_fbFileClose(
	sNetId:= , 
	hFile:=_fbFileOpen.hFile , 
	bExecute:= , 
	tTimeout:= , 
	bBusy=> , 
	bError=> , 
	nErrId=> );
	
A_Run();
A_Status();

ACTION A_Run:
{attribute'hide'}

IF NOT Execute THEN
	_iRun:=0;
END_IF

CASE _iRun OF
	0:
		Done:=FALSE;
		_fbFileOpen.bExecute:=FALSE;
		_fbFileClose.bExecute:=FALSE;
		_fbFileWrite.bExecute:=FALSE;
		IF Execute THEN
			_iRun:=100;
		END_IF
	100:
		_fbFileOpen.bExecute:=TRUE;
		IF _fbFileOpen.bBusy THEN
			_iRun:=200;
		END_IF
	200:
		IF NOT _fbFileOpen.bBusy  THEN
			_fbFileOpen.bExecute:=FALSE;
			_iRun:=300;
		END_IF

	300:
		_fbFileWrite.bExecute:=TRUE;
		IF _fbFileWrite.bBusy  THEN
			_iRun:=400;
		END_IF
	400:
		IF NOT _fbFileWrite.bBusy THEN
			_fbFileWrite.bExecute:=FALSE;
			_iRun:=500;
		END_IF
	500:
		_fbFileClose.bExecute:=TRUE;
		IF _fbFileClose.bBusy  THEN
			_iRun:=600;
		END_IF
	600:
		IF NOT _fbFileClose.bBusy THEN
			_fbFileClose.bExecute:=FALSE;
			_iRun:=700;
		END_IF
	700:
		Done:=TRUE;
		IF NOT Execute  THEN
			_iRun:=0;
		END_IF
END_CASE
END_ACTION

ACTION A_Status:
{attribute'hide'}

Busy:= _fbFileOpen.bBusy  OR _fbFileWrite.bBusy OR _fbFileClose.bBusy;

Error:=_fbFileOpen.bError OR _fbFileWrite.bError OR _fbFileClose.bError;
END_ACTION

END_FUNCTION_BLOCK

// File/POUs/FB_LogHelper_B
FUNCTION_BLOCK FB_LogHelper_B // 带缓存功能的Log文件写入
VAR_INPUT
	System:						REFERENCE TO ST_System;
	FliePath:					STRING;// 文件夹路径					
	Message:					WSTRING(255);// 写入信息
END_VAR
VAR_OUTPUT
END_VAR
VAR
	_fbFileLog:					FB_LogHelper;
	_fbFifo:					FB_MemRingBuffer;
	_sFifoWrite:				WSTRING(255);
	_sFifoRead:					WSTRING(255);
	_arrFifoBuffer:				ARRAY[0..1000] OF WSTRING(255);
	_iFifoCount:				UDINT;
	_tonWrite:					TON;
	_fbDirectoryHelper:			FB_DirectoryHelper1;
END_VAR

IF _fbFifo.nCount>0 AND NOT _fbFileLog.Execute  AND NOT _fbFileLog.Done  AND NOT _tonWrite.Q THEN
	_sFifoRead:="";
	_iFifoCount:=_fbFifo.nCount;
	_fbFifo.A_RemoveHead();
	_fbFileLog.Message:=_sFifoRead;
	_fbFileLog.Execute:=TRUE;
END_IF
IF  _fbFileLog.Done OR _fbFileLog.Error THEN
	_fbFileLog.Execute:=FALSE;
END_IF


_fbDirectoryHelper(
	Execute:=TRUE , 
	Command:=E_Directory.Create , 
	FolderPath:=FliePath , 
	Busy=> , 
	Error=> , 
	Done=> );

_fbFileLog(
	Execute:= , 
	FilePath:=CONCAT(CONCAT(CONCAT(FliePath,'\'),System.stSystemDate.sDateDay),'.txt') , 
	Message:= , 
	Done=> , 
	Busy=> , 
	Error=> , 
	ErrId=> );
	
_fbFifo(
	pWrite:=ADR(_sFifoWrite) , 
	cbWrite:=SIZEOF(_sFifoWrite) , 
	pRead:=ADR(_sFifoRead) , 
	cbRead:=SIZEOF(_sFifoRead) , 
	pBuffer:=ADR(_arrFifoBuffer) , 
	cbBuffer:=SIZEOF(_arrFifoBuffer) , 
	bOk=> , 
	nCount=> , 
	cbSize=> , 
	cbReturn=> );
	
_tonWrite(IN:=_fbFifo.nCount=_iFifoCount AND NOT _fbFifo.nCount<>0  , PT:=T#2S , Q=> , ET=> );

ACTION A_AddTail:
_sFifoWrite:=Message;
_fbFifo.A_AddTail();
END_ACTION

END_FUNCTION_BLOCK

// File/POUs/FB_LogHelper_E
FUNCTION_BLOCK FB_LogHelper_E// 英文Log文件写入
VAR_INPUT
	Execute:				BOOL;
	FilePath:				STRING;
	Message:				STRING(1000);
END_VAR
VAR_OUTPUT
	Done:					BOOL;
	Busy:					BOOL;
	Error:					BOOL;
	ErrId:					INT;// 暂未使用
END_VAR
VAR
	_iRun:					INT;
	_fbFileOpen:			FB_FileOpen;
	_fbFileWrite:			FB_FileWrite;
	_fbFileClose:			FB_FileClose;
	_sTempString:			STRING(1000);
	_arrTemp:				ARRAY[0..1] OF STRING(1000);
	_sSeparator:			STRING;
END_VAR

_fbFileOpen(
	sNetId:= , 
	sPathName:=FilePath , 
	nMode:=FOPEN_MODEAPPEND , 
	ePath:= , 
	bExecute:= , 
	tTimeout:= , 
	bBusy=> , 
	bError=> , 
	nErrId=> , 
	hFile=> );

_arrTemp[0]:=Message;
_arrTemp[1]:='$N';
_sTempString:=F_Join_L(ADR(_arrTemp),SIZEOF(_arrTemp[0]),1,ADR(_sSeparator),SIZEOF(_sSeparator));

_fbFileWrite(
	sNetId:= , 
	hFile:=_fbFileOpen.hFile , 
	pWriteBuff:=ADR(_sTempString) , 
	cbWriteLen:=F_LEN(ADR(_sTempString)), 
	bExecute:= , 
	tTimeout:= , 
	bBusy=> , 
	bError=> , 
	nErrId=> , 
	cbWrite=> );

_fbFileClose(
	sNetId:= , 
	hFile:=_fbFileOpen.hFile , 
	bExecute:= , 
	tTimeout:= , 
	bBusy=> , 
	bError=> , 
	nErrId=> );
	
A_Run();
A_Status();

ACTION A_Run:
{attribute'hide'}

IF NOT Execute THEN
	_iRun:=0;
END_IF

CASE _iRun OF
	0:
		Done:=FALSE;
		_fbFileOpen.bExecute:=FALSE;
		_fbFileClose.bExecute:=FALSE;
		_fbFileWrite.bExecute:=FALSE;
		IF Execute THEN
			_iRun:=100;
		END_IF
	100:
		_fbFileOpen.bExecute:=TRUE;
		IF _fbFileOpen.bBusy THEN
			_iRun:=200;
		END_IF
	200:
		IF NOT _fbFileOpen.bBusy  THEN
			_fbFileOpen.bExecute:=FALSE;
			_iRun:=300;
		END_IF

	300:
		_fbFileWrite.bExecute:=TRUE;
		IF _fbFileWrite.bBusy  THEN
			_iRun:=400;
		END_IF
	400:
		IF NOT _fbFileWrite.bBusy THEN
			_fbFileWrite.bExecute:=FALSE;
			_iRun:=500;
		END_IF
	500:
		_fbFileClose.bExecute:=TRUE;
		IF _fbFileClose.bBusy  THEN
			_iRun:=600;
		END_IF
	600:
		IF NOT _fbFileClose.bBusy THEN
			_fbFileClose.bExecute:=FALSE;
			_iRun:=700;
		END_IF
	700:
		Done:=TRUE;
		IF NOT Execute  THEN
			_iRun:=0;
		END_IF
END_CASE
END_ACTION

ACTION A_Status:
{attribute'hide'}

Busy:= _fbFileOpen.bBusy  OR _fbFileWrite.bBusy OR _fbFileClose.bBusy;

Error:=_fbFileOpen.bError OR _fbFileWrite.bError OR _fbFileClose.bError;
END_ACTION

END_FUNCTION_BLOCK

// Regex/F_Join_L
FUNCTION F_Join_L:STRING(2000)
VAR_INPUT
	In:						POINTER TO BYTE;// 拼接字符串数组
	OneLength:				UDINT;//Sizeof(In[0])
	Count:					INT;// 数组长度
	Separator:				POINTER TO BYTE;// 分隔符
	SeparatorLength:		UDINT;//Sizeof(SeparatorLength)
END_VAR
VAR
	_i:						LINT;// 输入字符串数组循环
	_t:						LINT;// 单个输入字符串循环
	_f:						LINT;// 输出元素索引
	_a:						LINT;// 
	_pTemp:					POINTER TO BYTE;
	_iTemplen:				UINT;
END_VAR

_pTemp:=ADR(F_Join_L);
_iTemplen:=SIZEOF(F_Join_L);

FOR _i:=0 TO Count BY 1 DO
	FOR _t:=(_i*OneLength) TO (OneLength-1)+(OneLength*_i) BY 1 DO
		IF _f>=_iTemplen-1 THEN RETURN; END_IF;
		IF In[_t]=0 THEN EXIT; END_IF;
		_pTemp[_f]:=In[_t];
		_f:=_f+1;
	END_FOR
	IF _i=Count THEN
		EXIT;
	END_IF
	FOR _a:=0 TO SeparatorLength-1 BY 1 DO
		IF _f>=_iTemplen-1 THEN RETURN; END_IF;
		IF Separator[_a]=0 THEN EXIT; END_IF;
		_pTemp[_f]:=Separator[_a];
		_f:=_f+1;
	END_FOR
END_FOR
_pTemp[_f]:=0;

END_FUNCTION

// File/POUs/FB_LogHelper_E_B
FUNCTION_BLOCK FB_LogHelper_E_B// 英文带缓存的Log文件写入
VAR_INPUT
	System:						REFERENCE TO ST_System;
	DocumentPath:				STRING;// 文件夹路径					
	Message:					STRING(1000);// 写入信息
	FilePath:					STRING(1000);// 文件路径(当文件路径为空时 则按文件夹路路径自动生成文件)
END_VAR
VAR_OUTPUT
END_VAR
VAR
	_fbFileLog:					FB_LogHelper_E;
	_fbFifo:					FB_MemRingBuffer;
	_sFifoWrite:				STRING(1000);
	_sFifoRead:					STRING(1000);
	_arrFifoBuffer:				ARRAY[0..1000] OF STRING(1000);
	_iFifoCount:				UDINT;
	_tonWrite:					TON;
	_fbDirectoryHelper:			FB_DirectoryHelper;
END_VAR

IF _fbFifo.nCount>0 AND NOT _fbFileLog.Execute  AND NOT _fbFileLog.Done  AND NOT _tonWrite.Q THEN
	_sFifoRead:='';
	_iFifoCount:=_fbFifo.nCount;
	_fbFifo.A_RemoveHead();
	_fbFileLog.Message:=_sFifoRead;
	_fbFileLog.Execute:=TRUE;
END_IF
IF  _fbFileLog.Done OR _fbFileLog.Error THEN
	_fbFileLog.Execute:=FALSE;
END_IF

_fbDirectoryHelper(
	Execute:=TRUE , 
	Command:=E_Directory.Create , 
	DirectoryPath:=FilePath , 
	Busy=> , 
	Error=> , 
	Done=> );

_fbFileLog(
	Execute:= , 
	FilePath:=SEL(FilePath='',FilePath,CONCAT(CONCAT(CONCAT(DocumentPath,'\'),System.stSystemDate.sDateDay),'.txt')), 
	Message:= , 
	Done=> , 
	Busy=> , 
	Error=> , 
	ErrId=> );
	
_fbFifo(
	pWrite:=ADR(_sFifoWrite) , 
	cbWrite:=SIZEOF(_sFifoWrite) , 
	pRead:=ADR(_sFifoRead) , 
	cbRead:=SIZEOF(_sFifoRead) , 
	pBuffer:=ADR(_arrFifoBuffer) , 
	cbBuffer:=SIZEOF(_arrFifoBuffer) , 
	bOk=> , 
	nCount=> , 
	cbSize=> , 
	cbReturn=> );
	
_tonWrite(IN:=_fbFifo.nCount=_iFifoCount AND NOT _fbFifo.nCount<>0  , PT:=T#2S , Q=> , ET=> );

ACTION A_AddTail:
_sFifoWrite:=Message;
_fbFifo.A_AddTail();
END_ACTION

END_FUNCTION_BLOCK

// File/POUs/FB_LogHelper1
FUNCTION_BLOCK FB_LogHelper1
VAR_INPUT
	FilePath:				STRING;// 文件路径
	pBuffer:				PVOID;// 缓存数据区
	cbBuffer:				UDINT;// sizfof(cbBuffer)
	Message:				PVOID;// 写入信息
END_VAR
VAR_OUTPUT
END_VAR
VAR
	_sFifoRead:				STRING(1000);
	_iFifoCount:			UDINT;
	_fbFileHelper:			FB_FileHelper;
	_fbFifo:				FB_MemRingBuffer;
END_VAR

_fbFifo(
	pWrite:= , 
	cbWrite:= , 
	pRead:=ADR(_sFifoRead) , 
	cbRead:=SIZEOF(_sFifoRead) , 
	pBuffer:=pBuffer , 
	cbBuffer:=cbBuffer , 
	bOk=> , 
	nCount=> , 
	cbSize=> , 
	cbReturn=> );
_fbFileHelper(
	Read:= , 
	WriteAllText:= , 
	AppendAllText:= , 
	FilePath:=FilePath , 
	Buffer:=ADR(_sFifoRead) , 
	BufferLen:=F_LEN(ADR(_sFifoRead)) , 
	TimeOut:= , 
	Busy=> , 
	Error=> , 
	Done=> );
	
	
IF _fbFifo.nCount>0 AND NOT _fbFileHelper.AppendAllText THEN
	_sFifoRead:='';
	_fbFifo.A_RemoveHead();
	_fbFileHelper.AppendAllText:=TRUE;
END_IF
IF  _fbFileHelper.Done THEN
	_fbFileHelper.AppendAllText:=FALSE;
END_IF

METHOD M_AddTail : BOOL
VAR_INPUT
END_VAR
_fbFifo.pWrite:=Message;
_fbFifo.cbWrite:=F_LEN(Message);
_fbFifo.A_AddTail();
M_AddTail:=TRUE;
END_METHOD

END_FUNCTION_BLOCK

// Hive/POUs/FB_Hive
FUNCTION_BLOCK FB_Hive
VAR_INPUT
	System:				 	 REFERENCE TO ST_System;
	Error:				  	 REFERENCE TO ST_Error;
	Hive:					 REFERENCE TO ST_Hive;
	Data:					 REFERENCE TO ST_HiveData;
END_VAR
VAR_OUTPUT
END_VAR
VAR
	_arrFbHttpClient:		ARRAY[0..3] OF FB_HttpClient;
	_arrHttpClient:			ARRAY[0..3] OF ST_HttpClient;
	_arrHttpClientData:		ARRAY[0..3] OF ST_HttpClientData;
	_i:						INT;
	_eHiveState:			E_HiveState:=E_HiveState.None;
	_iStateRun:				INT;
	_iDataRun:				INT;
	_sDataTime:				STRING;
	
	_arrErrorTemp:			ARRAY[0..100] OF STRING;
	_arrErrorCode:			ARRAY[0..100] OF STRING;
	_arrErrorMessage:		ARRAY[0..100] OF STRING;
	_iErrorCount:			INT:=0;
	_sErrorMessageTemp:		STRING(1000);
	
	_arrTon:				ARRAY[0..10] OF TON;
	
	_iRunCount:				INT:=0;
	
	_iModeRun:				INT;
	_bFirstRun:				BOOL:=TRUE;
END_VAR

IF _iRunCount<3 THEN
	_iRunCount:=_iRunCount+1;
	RETURN;
END_IF
IF  _bFirstRun THEN
	A_Init();
END_IF



IF Hive.stControl.bDataEnable THEN
	_arrFbHttpClient[0](System:=System , Error:=Error , HttpClient:=_arrHttpClient[0] , Data:=_arrHttpClientData[0] );
END_IF

IF Hive.stControl.bDataEnable THEN
	_arrFbHttpClient[1](System:=System , Error:=Error , HttpClient:=_arrHttpClient[1] , Data:=_arrHttpClientData[1] );
END_IF

IF Hive.stControl.bStateEnable THEN
	_arrFbHttpClient[2](System:=System , Error:=Error , HttpClient:=_arrHttpClient[2] , Data:=_arrHttpClientData[2] );
END_IF

IF Hive.stControl.bDataEnable THEN
	_arrFbHttpClient[3](System:=System , Error:=Error , HttpClient:=_arrHttpClient[3] , Data:=_arrHttpClientData[3] );
END_IF



//2020-08-27T00:01:29.51+0800
_sDataTime:=M_DateTime();
A_Data();
A_Mode();
A_State();
A_Ton();

_bFirstRun:=FALSE;

ACTION A_Data:
{attribute'hide'}

IF System.stInput.bReset OR NOT  Hive.stControl.bDataEnable THEN
	_iDataRun:=0;
END_IF

CASE _iDataRun OF
	0:
		Hive.stSendDataState.bDone:=FALSE;
		Hive.stSendDataState.bBusy:=FALSE;
		Hive.stSendDataState.bError:=FALSE;
		_arrHttpClient[0].stControl.eRequest:=E_HttpRequestOrder.None;
		IF Hive.stControl.bSendData AND Hive.stControl.bDataEnable THEN
			_iDataRun:=100;
		END_IF;
	100:
		Hive.stSendDataState.bBusy:=TRUE;
		_arrHttpClient[0].stControl.sRequestData:=M_Data();
		_iDataRun:=200;
	200:
		_arrHttpClient[0].stControl.eRequest:=E_HttpRequestOrder.POST;
		IF _arrHttpClient[0].stStatus.bDone OR _arrTon[2].Q  THEN
			_arrHttpClient[0].stControl.eRequest:=E_HttpRequestOrder.None;
			_iDataRun:=300;
		END_IF
	300:
		IF  _arrTon[2].Q THEN
			Hive.stSendDataState.bError:=TRUE;
		END_IF;
		_iDataRun:=400;
	400:
		Hive.stSendDataState.bBusy:=FALSE;
		Hive.stSendDataState.bDone:=TRUE;
		IF NOT  Hive.stControl.bSendData AND NOT System.stMode.bStop THEN
			Hive.stSendDataState.bDone:=FALSE;
			_iDataRun:=0;
		END_IF
END_CASE
END_ACTION

ACTION A_Init:
{attribute'hide'}

_arrHttpClient[0].arrInfo[E_Language.Chinese].sName:="Hive_Data";
_arrHttpClient[0].arrInfo[E_Language.English].sName:="Hive_Data";
_arrHttpClient[0].arrInfo[E_Language.Hindi].sName:="Hive_Data";
_arrHttpClient[0].arrInfo[E_Language.Vietnamese].sName:="Hive_Data";
_arrHttpClientData[0].iPort:=Data.stDataAddress.iPort;
_arrHttpClientData[0].iTimeOut:=Data.iTimeOut;
_arrHttpClientData[0].sIP:=Data.stDataAddress.sIP;
_arrHttpClientData[0].sUri:=Data.stDataAddress.sUri;

_arrHttpClient[1].arrInfo[E_Language.Chinese].sName:="Hive_Mode";
_arrHttpClient[1].arrInfo[E_Language.English].sName:="Hive_Mode";
_arrHttpClient[1].arrInfo[E_Language.Hindi].sName:="Hive_Mode";
_arrHttpClient[1].arrInfo[E_Language.Vietnamese].sName:="Hive_Mode";
_arrHttpClientData[1].iPort:=Data.stModeAddressOn.iPort;
_arrHttpClientData[1].iTimeOut:=Data.iTimeOut;
_arrHttpClientData[1].sIP:=Data.stModeAddressOn.sIP;
_arrHttpClientData[1].sUri:=Data.stModeAddressOn.sUri;

_arrHttpClient[2].arrInfo[E_Language.Chinese].sName:="Hive_State";
_arrHttpClient[2].arrInfo[E_Language.English].sName:="Hive_State";
_arrHttpClient[2].arrInfo[E_Language.Hindi].sName:="Hive_State";
_arrHttpClient[2].arrInfo[E_Language.Vietnamese].sName:="Hive_State";
_arrHttpClientData[2].iPort:=Data.stStateAddress.iPort;
_arrHttpClientData[2].iTimeOut:=Data.iTimeOut;
_arrHttpClientData[2].sIP:=Data.stStateAddress.sIP;
_arrHttpClientData[2].sUri:=Data.stStateAddress.sUri;

_arrHttpClient[3].arrInfo[E_Language.Chinese].sName:="Hive_Mode";
_arrHttpClient[3].arrInfo[E_Language.English].sName:="Hive_Mode";
_arrHttpClient[3].arrInfo[E_Language.Hindi].sName:="Hive_Mode";
_arrHttpClient[3].arrInfo[E_Language.Vietnamese].sName:="Hive_Mode";
_arrHttpClientData[3].iPort:=Data.stModeAddressOff.iPort;
_arrHttpClientData[3].iTimeOut:=Data.iTimeOut;
_arrHttpClientData[3].sIP:=Data.stModeAddressOff.sIP;
_arrHttpClientData[3].sUri:=Data.stModeAddressOff.sUri;
END_ACTION

ACTION A_Mode:
{attribute'hide'}

IF  _arrTon[3].Q OR _arrTon[4].Q THEN
	_iModeRun:=0;
END_IF

CASE _iModeRun OF
	0:
		_arrTon[3].IN:=_arrTon[4].IN:=FALSE;
		_arrHttpClient[1].stControl.eRequest:=E_HttpRequestOrder.None;
		_arrHttpClient[3].stControl.eRequest:=E_HttpRequestOrder.None;
		IF Hive.stControl.bModeLogin AND Hive.stControl.bModeEnable THEN
			_iModeRun:=100;
		END_IF
	100:
		_arrHttpClient[1].stControl.sRequestData:=M_ModeOn();
		_iModeRun:=200;
	200:
		_arrTon[3].IN:=TRUE;
		_arrHttpClient[1].stControl.eRequest:=E_HttpRequestOrder.POST;
		IF _arrHttpClient[1].stStatus.bDone THEN
			_arrHttpClient[1].stControl.eRequest:=E_HttpRequestOrder.None;
			_iModeRun:=300;
		END_IF
	300:
		IF NOT Hive.stControl.bModeLogin THEN
			_iModeRun:=400;
		END_IF
	400:
		_arrHttpClient[3].stControl.sRequestData:=M_ModeOff();
		_iModeRun:=500;
	500:
		_arrTon[4].IN:=TRUE;
		_arrHttpClient[3].stControl.eRequest:=E_HttpRequestOrder.POST;
		IF _arrHttpClient[3].stStatus.bDone THEN
			_arrHttpClient[3].stControl.eRequest:=E_HttpRequestOrder.None;
			_iModeRun:=0;
		END_IF
END_CASE
END_ACTION

ACTION A_State:
{attribute'hide'}

IF System.stMode.bAutoRunning OR System.stMode.bHoming THEN
	_eHiveState:=E_HiveState.Running;
END_IF;

IF System.stMode.bIdle OR System.stMode.bNone THEN
	_eHiveState:=E_HiveState.Idle;
END_IF;

IF System.stMode.arrAlarm[1] OR  System.stMode.arrAlarm[2] OR System.stMode.arrAlarm[3] THEN
	_eHiveState:=E_HiveState.UnplannedDown;
END_IF;

IF System.stMode.bManual THEN
	_eHiveState:=E_HiveState.Engineering;
END_IF;

IF Hive.stControl.bPlannedDown THEN
	_eHiveState:=E_HiveState.PlannedDown;
END_IF;


IF _arrTon[1].Q OR NOT Hive.stControl.bStateEnable THEN
	_iStateRun:=0;
END_IF; 

CASE _iStateRun OF
	0:
		_arrTon[0].IN:=FALSE;
		_arrHttpClient[2].stControl.eRequest:=E_HttpRequestOrder.None;
		IF _eHiveState <> Hive.eState AND Hive.stControl.bStateEnable AND NOT _arrTon[1].Q THEN
			_iStateRun:=100;
		END_IF;
	100:
		CASE _eHiveState OF
			0:
				_iStateRun:=0;
			1,2,3,4:
				_iStateRun:=200;
			5:
				_iStateRun:=500;
		END_CASE
	200:
		_arrHttpClient[2].stControl.sRequestData:=M_State(_eHiveState,'');
		_iStateRun:=1000;
	500:
		FOR _i:=0 TO 100 BY 1 DO
			_arrErrorTemp[_i]:='';
			_arrErrorCode[_i]:='';
			_arrErrorMessage[_i]:='';
			_iErrorCount:=0;
		END_FOR
		_iStateRun:=510;
	510:// 报警信息为: 报警文本;报警代码
		FOR _i:=0 TO Error.stNow.iCount BY 1 DO
			IF STRING_TO_INT(Error.stNow.arrInfo[_i].sLevel)<=3 AND Error.stNow.arrInfo[_i].sLevel<>'' THEN
				_sErrorMessageTemp:=WSTRING_TO_STRING(Error.stNow.arrInfo[_i].arrMessage[Data.eLanguage]);
				F_Split(ADR(_sErrorMessageTemp),ADR(';'),ADR(_arrErrorTemp),SIZEOF(_arrErrorTemp[0]),SIZEOF(_arrErrorTemp));
				EXIT;
			END_IF
		END_FOR
		_iStateRun:=515;
	515:
		_arrErrorMessage[_iErrorCount]:=_arrErrorTemp[0];
		_arrErrorCode[_iErrorCount]:=_arrErrorTemp[1];
		_iStateRun:=520;
	520:
		_arrErrorTemp[0]:=CONCAT(CONCAT(CONCAT(CONCAT(CONCAT('$R"code": "',_arrErrorCode[_iErrorCount]),'",'),'$R"error_message" : "'),_arrErrorMessage[_iErrorCount]),'",$R');
		_arrHttpClient[2].stControl.sRequestData:=M_State(_eHiveState,_arrErrorTemp[0]);
		_iErrorCount:=_iErrorCount+1;
		_iStateRun:=1000;
	1000:
		_arrTon[0].IN:=TRUE;
		_arrHttpClient[2].stControl.eRequest:=E_HttpRequestOrder.POST;
		IF _arrHttpClient[2].stStatus.bDone THEN
			_arrHttpClient[2].stControl.eRequest:=E_HttpRequestOrder.None;
			_iStateRun:=1100;
		END_IF
	1100:
		IF NOT _arrTon[0].Q THEN
			 Hive.eState:=_eHiveState;
		END_IF
		_iStateRun:=0;
END_CASE
END_ACTION

ACTION A_Ton:
{attribute'hide'}

_arrTon[0](IN:= , PT:=UINT_TO_TIME(Data.iTimeOut) , Q=> , ET=> );// State处理耗时
_arrTon[1](IN:= _iStateRun<>0, PT:=UINT_TO_TIME(Data.iTimeOut+1000), Q=> , ET=> );// State运行耗时

_arrTon[2](IN:=Hive.stSendDataState.bBusy , PT:=UINT_TO_TIME(Data.iTimeOut+500) , Q=> , ET=> );// Data处理耗时

_arrTon[3](IN:= , PT:=UINT_TO_TIME(Data.iTimeOut+500) , Q=> , ET=> );//ModeOn处理耗时
_arrTon[4](IN:= , PT:=UINT_TO_TIME(Data.iTimeOut+500) , Q=> , ET=> );//ModeOff处理耗时
END_ACTION

{attribute'hide'}
METHOD M_Data : STRING(2000)
VAR_INPUT
END_VAR
VAR
	_t:						INT;
	_arrTemp:				ARRAY[0..400] OF STRING;
	_iCount:				INT;
	_temp:					POINTER TO BYTE;
END_VAR


_arrTemp[0]:='{';
_arrTemp[1]:=CONCAT(CONCAT('"unit_sn": "',Hive.stControl.stMachineData.sUnit_sn),'",');
_arrTemp[2]:='"serials": {';
_arrTemp[3]:=CONCAT(CONCAT('"carrier_sn": "',Hive.stControl.stMachineData.sCarrier_sn),'",');
_arrTemp[4]:=CONCAT(CONCAT('"wip_serials" : ["',Hive.stControl.stMachineData.sWip_serials),'"]},');
_arrTemp[5]:=CONCAT(CONCAT('"pass": "',BOOL_TO_STRING( Hive.stControl.stMachineData.bPass)),'",');
_arrTemp[6]:=CONCAT(CONCAT('"input_time": "',Hive.stControl.stMachineData.sInput_time),'",');
_arrTemp[7]:=CONCAT(CONCAT('"output_time": "',Hive.stControl.stMachineData.sOutput_time),'",');
_arrTemp[8]:='"data": {';
_iCount:=8;
FOR _t:=0 TO Hive.stControl.stMachineData.iDataCount-1 BY 1 DO
	IF Hive.stControl.stMachineData.arrDataName[_t]<>'' THEN
		_arrTemp[9+_t]:=CONCAT(CONCAT(CONCAT(CONCAT('"',Hive.stControl.stMachineData.arrDataName[_t]),'":"'),Hive.stControl.stMachineData.arrDataValue[_t]),'",');
		_iCount:=_iCount+1;
	END_IF;
END_FOR
IF _iCount>8 THEN
	_temp:=ADR(_arrTemp[_iCount]);
	_temp[F_LEN(ADR(_arrTemp[_iCount]))-1]:=0;
END_IF
_arrTemp[_iCount+1]:='}$R}';

M_Data:=F_Join_L(ADR(_arrTemp),SIZEOF(_arrTemp[0]),_iCount+1,ADR('$R'),SIZEOF('$R'));
END_METHOD

{attribute'hide'}
METHOD M_DateTime : string
VAR_INPUT
END_VAR


M_DateTime:=CONCAT(CONCAT(CONCAT(CONCAT(CONCAT(CONCAT(CONCAT(CONCAT(CONCAT(CONCAT(CONCAT(CONCAT(CONCAT(CONCAT(INT_TO_STRING(System.stSystemDate.iYear),'-'),M_Join0(system.stSystemDate.iMonth)),'-'),M_Join0(system.stSystemDate.iDay)),'T'),M_Join0(system.stSystemDate.iHour)),':'),M_Join0(system.stSystemDate.iMinute)),':'),M_Join0(system.stSystemDate.iSecond)),'.'),INT_TO_STRING(System.stSystemDate.iMilliseconds)),'+'),'0800');
END_METHOD

{attribute'hide'}
METHOD M_Join0 : STRING
VAR_INPUT
	In:					INT;
END_VAR


M_Join0:=SEL(In<10,INT_TO_STRING(In),CONCAT('0',INT_TO_STRING(In)));
END_METHOD

{attribute'hide'}
METHOD M_ModeOff : STRING(2000)
VAR_INPUT
END_VAR
VAR
	_arrTemp:				ARRAY[0..2] OF STRING(1000);
	_arrTemp1:				ARRAY[0..100] OF STRING;
	_iCount:				INT:=0;
	_t:						INT;
END_VAR


FOR _t:=0 TO Hive.stControl.iActivityCount-1 BY 1 DO
	IF Hive.stControl.arrActivity[_t]<>'' THEN
		_arrTemp1[_t]:=CONCAT(CONCAT('"', Hive.stControl.arrActivity[_t]),'"');
		_iCount:=_iCount+1;
	END_IF
END_FOR

_arrTemp[0]:=CONCAT(CONCAT('{$R"state_time": "',_sDataTime),'",$R"data": {$R"activity" : [');
_arrTemp[1]:=F_Join_L(ADR(_arrTemp1),SIZEOF(_arrTemp1[0]),_iCount-1,ADR(','),SIZEOF(','));;
_arrTemp[2]:= CONCAT(CONCAT('],$R"session_token": "',Hive.stControl.sSession_token),'"$R}$R}');


M_ModeOff:=F_Join_L(ADR(_arrTemp),SIZEOF(_arrTemp[0]),2,ADR('$R'),SIZEOF('$R'));
END_METHOD

{attribute'hide'}
METHOD M_ModeOn : STRING(2000)
VAR_INPUT
END_VAR
VAR
	_arrTemp:				ARRAY[0..10] OF STRING(100);
END_VAR


_arrTemp[0]:='{';
_arrTemp[1]:=CONCAT(CONCAT('"state_time": "',_sDataTime),'",');
_arrTemp[2]:='"data": {';
_arrTemp[3]:= CONCAT(CONCAT('"session_token": "',Hive.stControl.sSession_token),'"');
_arrTemp[4]:='}';
_arrTemp[5]:='}';

M_ModeOn:=F_Join_L(ADR(_arrTemp),SIZEOF(_arrTemp[0]),5,ADR('$R'),SIZEOF('$R'));
END_METHOD

{attribute'hide'}
METHOD M_State : STRING(2000)
VAR_INPUT
	State:					INT;
	Data:					STRING(1000);
END_VAR
VAR
	_arrTemp:				ARRAY[0..100] OF STRING(255);
END_VAR


_arrTemp[0]:='{';
_arrTemp[1]:=CONCAT(CONCAT('"machine_state":',INT_TO_STRING(State)),',');
_arrTemp[2]:=CONCAT(CONCAT('"state_change_time": "',_sDataTime),'",');
_arrTemp[3]:=CONCAT(CONCAT('"data": {',Data),'}');
_arrTemp[4]:='}';
M_State:=F_Join_L(ADR(_arrTemp),SIZEOF(_arrTemp[0]),4,ADR('$R'),SIZEOF('$R'));
END_METHOD

END_FUNCTION_BLOCK

// Http/POUs/FB_HttpClient
FUNCTION_BLOCK FB_HttpClient
VAR_INPUT
	System:						REFERENCE TO ST_System;
	Error:						REFERENCE TO ST_Error;
	HttpClient:					REFERENCE TO ST_HttpClient;
	Data:						REFERENCE TO ST_HttpClientData;
END_VAR
VAR_OUTPUT
END_VAR
VAR
	_fbIotHttpClient:					FB_IotHttpClient();
	_fbIotHttpRequest:					FB_IotHttpRequest();
	_fbIotHttpHeaderFieldMap:			FB_IotHttpHeaderFieldMap();
	_run:								INT;
	_arrFbErrorTag:						ARRAY[0..2] OF FB_ErrorTag;
	_i:									INT;
	_bFistRun:							BOOL:=TRUE;
END_VAR

HttpClient.sName:=HttpClient.arrInfo[System.stMode.eLanguage].sName;

_fbIotHttpClient.sHostName:=Data.sIP;
_fbIotHttpClient.nHostPort:=Data.iPort;
_fbIotHttpClient.Execute();

IF System.stInput.bReset THEN
	HttpClient.stControl.eRequest:=E_HttpRequestOrder.None;
	_run:=0;
END_IF;

IF _bFistRun THEN
	A_Init();
END_IF

A_Run();

A_Error();

_bFistRun:=FALSE;

ACTION A_Error:
{attribute'hide'}

_arrFbErrorTag[0](
	System:=System , 
	Error:=Error , 
	Enable:=_fbIotHttpClient.bError OR _fbIotHttpRequest.bError OR _fbIotHttpHeaderFieldMap.bError , 
	Message:=, 
	Level:=5 , 
	Position:=WCONCAT("FB_HttpClient:",HttpClient.arrInfo[E_Language.Chinese].sName) , 
	ErrorTime:= , 
	Language:= , 
	Erroring=>HttpClient.stStatus.bError,
	ID:=HttpClient.ID,
	Category:=E_ErrorCategory.Http,
	InfoIndex:=0);

	
_arrFbErrorTag[1](
	System:=System , 
	Error:=Error , 
	Enable:=HttpClient.stStatus.bBusy, 
	Message:="Http通信超时" , 
	Level:=5 , 
	Position:=WCONCAT("FB_HttpClient:",HttpClient.arrInfo[E_Language.Chinese].sName) , 
	ErrorTime:=UINT_TO_TIME(Data.iTimeOut), 
	Language:= , 
	Erroring=> HttpClient.stStatus.bErrorTimeOut,
	ID:=HttpClient.ID,
	Category:=E_ErrorCategory.Http,
	InfoIndex:=1);
END_ACTION

ACTION A_Init:
{attribute'hide'}
	HttpClient.arrInfo[E_Language.Chinese].sError:="状态错误";
	HttpClient.arrInfo[E_Language.Chinese].sErrorTimeOut:="请求超时";
	
	HttpClient.arrInfo[E_Language.English].sError:="Status error";
	HttpClient.arrInfo[E_Language.English].sErrorTimeOut:="Request timeout";
	
	HttpClient.arrInfo[E_Language.Hindi].sError:="स्थिति गलत है";
	HttpClient.arrInfo[E_Language.Hindi].sErrorTimeOut:="अनुरोध समय पर बाहर";
	
	HttpClient.arrInfo[E_Language.Vietnamese].sError:="Lỗi trạng thái";
	HttpClient.arrInfo[E_Language.Vietnamese].sErrorTimeOut:="Yêu cầu thời gian chờ";

FOR _i:=0 TO E_Language.MaxCount BY 1 DO
	_arrFbErrorTag[0].Language[_i]:= WCONCAT(HttpClient.arrInfo[_i].sName,HttpClient.arrInfo[_i].sError);
	_arrFbErrorTag[1].Language[_i]:= WCONCAT(HttpClient.arrInfo[_i].sName,HttpClient.arrInfo[_i].sErrorTimeOut);
END_FOR;
END_ACTION

ACTION A_Run:
{attribute'hide'}

CASE _run OF
	0:
		HttpClient.stStatus.bBusy:=HttpClient.stStatus.bDone:=FALSE;
		IF HttpClient.stControl.eRequest<>E_HttpRequestOrder.None AND  NOT System.stMode.bStop THEN
			_run:=100;
		END_IF;
	100:
		HttpClient.stStatus.bBusy:=TRUE;
		CASE HttpClient.stControl.eRequest  OF
			E_HttpRequestOrder.GET:
				IF SendRequest(ETcIotHttpRequestType.HTTP_GET) THEN
					_run:=1000;
				END_IF
			E_HttpRequestOrder.POST:
				IF SendRequest(ETcIotHttpRequestType.HTTP_POST) THEN
					_run:=1000;
				END_IF
		END_CASE
	1000:
		IF NOT _fbIotHttpRequest.bBusy THEN
			HttpClient.stControl.sResponseData:='';
			_run:=1100;
		END_IF
	1100:
		IF _fbIotHttpRequest.nContentSize<>0 THEN
			_fbIotHttpRequest.GetContent(ADR(HttpClient.stControl.sResponseData),SIZEOF(HttpClient.stControl.sResponseData),TRUE);
		END_IF;
		_run:=1200;
	1200:
		HttpClient.stStatus.bBusy:=FALSE;
		HttpClient.stStatus.bDone:=TRUE;
		IF HttpClient.stControl.eRequest=E_HttpRequestOrder.None THEN
			HttpClient.stStatus.bDone:=FALSE;
			_run:=0;
		END_IF
END_CASE
END_ACTION

{attribute'hide'}
METHOD SendRequest : BOOL
VAR_INPUT
	 eRequestType : ETcIotHttpRequestType;
END_VAR
SendRequest:= _fbIotHttpRequest.SendRequest(sUri:=Data.sUri,fbClient:=_fbIotHttpClient,eRequestType:=eRequestType,pContent:=ADR(HttpClient.stControl.sRequestData),nContentSize:=F_LEN(ADR(HttpClient.stControl.sRequestData)),fbHeader:=_fbIotHttpHeaderFieldMap);
END_METHOD

END_FUNCTION_BLOCK

// Regex/F_Split
FUNCTION F_Split
VAR_INPUT
	In:							POINTER TO BYTE;// 要拆分的字符串
	Pattern:					POINTER TO BYTE;// 拆分规则
	Data:						POINTER TO BYTE;// 拆分分后 返回数组数据区
	OneLength:					UDINT;// Sizeof(Data[0])
	DataLength:					UDINT;// Sizeof(Data)
END_VAR
VAR
	_i:							LINT;// 拆分字符串 索引
	_t:							LINT;// 分隔符计数
	_tIdx:						LINT;// 分隔符位置 索引
	_f:							LINT;// 单个数据 索引
	_iLength:					LINT;// 分隔符与分割符 中间数据长度
	_tt:						LINT;// 分隔符计数
	_ttIdx:						LINT;// 分隔符位置 索引
	_iDataIdx:					LINT;// 数据数组 索引
	_x:							LINT;// 数据清空索引
	_y:							LINT;// 添加末尾数据索引
	_iPattern:					LINT;// 分隔符长度
	_idx:						LINT;// 末尾数据索引
	_bTemp:						BOOL;// 分隔符标志
END_VAR

FOR _x:=0 TO DataLength BY 1 DO
	Data[_x]:=0;
END_FOR
_iPattern:= F_LEN(Pattern);

WHILE In[_i]<> 0 DO
	WHILE _t<_iPattern AND In[_i]<> 0 DO
		_t:=SEL(In[_i]<>Pattern[_t],_t+1,0);
		_i:=_i+1;
	END_WHILE
	_bTemp:=_t>=_iPattern;
	_tIdx:=_i-1;
	FOR _f:=0 TO _iLength:=SEL(_ttIdx<>0,_tIdx-_ttIdx-1*_iPattern,_tIdx-_ttIdx-1*_iPattern-1) DO
		IF _iLength<0 OR _f>=OneLength OR NOT _bTemp THEN EXIT; END_IF;
		Data[_f+_iDataIdx*OneLength]:=In[SEL(_ttIdx<>0,_ttIdx+_f,_ttIdx+_f+1)];
	END_FOR
	IF In[_i]= 0 THEN EXIT; END_IF;
	_iDataIdx:=_iDataIdx+1;
	
	
	WHILE _tt<_iPattern AND In[_i]<> 0 DO
		_tt:=SEL(In[_i]<>Pattern[_tt],_tt+1,0);
		_i:=_i+1;
	END_WHILE
	_bTemp:=_tt>=_iPattern;
	_ttIdx:=_i-1;
	FOR _f:=0 TO _iLength:=_ttIdx-_tIdx-1*_iPattern-1 DO
		IF _iLength<0 OR _f>=OneLength OR NOT _bTemp THEN EXIT; END_IF;
		Data[_f+_iDataIdx*OneLength]:=In[_tIdx+_f+1];
	END_FOR
	IF In[_i]= 0 THEN EXIT; END_IF;
	_iDataIdx:=_iDataIdx+1;
	
	_t:=_tt:=0;
END_WHILE

IF _tIdx=0 AND _ttIdx=0 THEN
	FOR _y:=0 TO OneLength-1 BY 1 DO
		IF In[_y]=0 THEN EXIT; END_IF;
		Data[_y]:=In[_y];
	END_FOR
ELSIF NOT _bTemp THEN
	_idx:=SEL(_tIdx<_ttIdx,_ttIdx,_tIdx);
	FOR _y:=0 TO ABS(_tIdx-_ttIdx)-1 BY 1 DO
		Data[_y+_iDataIdx*OneLength]:=In[_idx+1+_y];
	END_FOR
END_IF

END_FUNCTION

// Regex/M_Join0
FUNCTION M_Join0 : String
VAR_INPUT
	In:				INT;
END_VAR
VAR
END_VAR

M_Join0:=SEL(In<10,INT_TO_STRING(In),CONCAT('0',INT_TO_STRING(In)));

END_FUNCTION

// Hive/POUs/P_Hive
PROGRAM P_Hive
VAR
END_VAR

METHOD M_Data : STRING(2000)
VAR_INPUT
	sUnit_sn:				STRING;
	sCarrier_sn:			STRING;
	sWip_serials:			STRING;
	sPass:					STRING;
	sInput_time:			STRING;
	sOutput_time:			STRING;
	arrDataName:			POINTER TO STRING;
	arrDataValue:			POINTER TO STRING;
	iDataCount:				UINT;
END_VAR
VAR
	_t:						UINT;
	_arrTemp:				ARRAY[0..10] OF STRING(255);
	_temp:					POINTER TO BYTE;
	_sData:					ARRAY[0..2] OF STRING(2000);
END_VAR
_arrTemp[0]:='{';
_arrTemp[1]:=CONCAT(CONCAT('"unit_sn": "',sUnit_sn),'",');
_arrTemp[2]:='"serials": {';
_arrTemp[3]:=CONCAT(CONCAT('"carrier_sn": "',sCarrier_sn),'",');
_arrTemp[4]:=CONCAT(CONCAT('"wip_serials" : [',sWip_serials),']},');
_arrTemp[5]:=CONCAT(CONCAT('"pass": "',sPass),'",');
_arrTemp[6]:=CONCAT(CONCAT('"input_time": "',sInput_time),'",');
_arrTemp[7]:=CONCAT(CONCAT('"output_time": "',sOutput_time),'",');
_arrTemp[8]:='"data": {';
_sData[0]:=F_Join_L(ADR(_arrTemp),SIZEOF(_arrTemp[0]),8,ADR(''),SIZEOF(''));
_sData[1]:=M_GetData(arrDataName,arrDataValue,iDataCount);
_sData[2]:='}}';
M_Data:=F_Join_L(ADR(_sData),SIZEOF(_sData[0]),2,ADR(''),SIZEOF(''));
END_METHOD

METHOD M_Error : String(2000)
VAR_INPUT
	Message:				STRING(1000);
	Code:					STRING;
	Occurrence_time:		STRING;
	Resolved_time:			STRING;
	arrDataName:			POINTER TO STRING;
	arrDataValue:			POINTER TO STRING;
	iDataCount:				UINT;
END_VAR
VAR
	_t:						UINT;
	_arrTemp:				ARRAY[0..10] OF STRING;
	_temp:					POINTER TO BYTE;
	_sData:					ARRAY[0..2] OF STRING(2000);
END_VAR
_sData[0]:='{"message":"';
_sData[1]:=Message;
_sData[2]:=F_Join_L(ADR(_sData),SIZEOF(_sData[0]),1,ADR(''),SIZEOF(''));
_sData[0]:=_sData[2];
_arrTemp[0]:='","code":"';
_arrTemp[1]:=Code;
_arrTemp[2]:='","';
_arrTemp[3]:='occurrence_time":"';
_arrTemp[4]:=Occurrence_time;
_arrTemp[5]:='","resolved_time":"';
_arrTemp[6]:=Resolved_time;
_arrTemp[7]:='","data":{';
_sData[1]:=F_Join_L(ADR(_arrTemp),SIZEOF(_arrTemp[0]),7,ADR(''),SIZEOF(''));
_sData[2]:='}}';
M_Error:=F_Join_L(ADR(_sData),SIZEOF(_sData[0]),2,ADR(''),SIZEOF(''));
END_METHOD

METHOD M_GetData : STRING(1000)
VAR_INPUT
	arrDataName:		POINTER TO STRING;
	arrDataValue:		POINTER TO STRING;
	iDataCount:			UINT;
END_VAR
VAR
	_t:					UINT;
	_iCount:			UINT;
	_arrTemp:			ARRAY[0..100] OF STRING;
	_temp:				POINTER TO BYTE;
END_VAR
IF iDataCount<=0 THEN RETURN; END_IF;

FOR _t:=0 TO iDataCount-1 BY 1 DO
	IF arrDataName[_t]<>'' THEN
		_arrTemp[_t]:=CONCAT(CONCAT(CONCAT(CONCAT('"',arrDataName[_t]),'":"'),arrDataValue[_t]),'",');
		_iCount:=_iCount+1;
	END_IF;
END_FOR
_temp:=ADR(_arrTemp[_iCount-1]);
_temp[F_LEN(ADR(_arrTemp[_iCount-1]))-1]:=0;

M_GetData:=F_Join_L(ADR(_arrTemp),SIZEOF(_arrTemp[0]),_iCount,ADR(''),SIZEOF(''));
END_METHOD

METHOD M_Mode : String(2000)
VAR_INPUT
	state_time:				STRING;
	arrDataName:			POINTER TO STRING;
	arrDataValue:			POINTER TO STRING;
	iDataCount:				UINT;
END_VAR
VAR
	_arrTemp:				ARRAY[0..10] OF STRING;
	_sData:					ARRAY[0..2] OF STRING(2000);
END_VAR
_arrTemp[0]:='{"state_time":"';
_arrTemp[1]:=state_time;
_arrTemp[2]:='","data":{';
_sData[0]:=F_Join_L(ADR(_arrTemp),SIZEOF(_arrTemp[0]),2,ADR(''),SIZEOF(''));
_sData[1]:=M_GetData(arrDataName,arrDataValue,iDataCount);
_sData[2]:='}}';
M_Mode:=F_Join_L(ADR(_sData),SIZEOF(_sData[0]),2,ADR(''),SIZEOF(''));
END_METHOD

METHOD M_State : STRING(2000)
VAR_INPUT
	State:					STRING;
	State_chage_time:		STRING;
	arrDataName:			POINTER TO STRING;
	arrDataValue:			POINTER TO STRING;
	iDataCount:				UINT;
END_VAR
VAR
	_arrTemp:				ARRAY[0..10] OF STRING(255);
	_iCount:				UINT;
	_sData:					ARRAY[0..3] OF STRING(1000);
END_VAR
_arrTemp[0]:='{';
_arrTemp[1]:=CONCAT(CONCAT('"machine_state":',State),',');
_arrTemp[2]:=CONCAT(CONCAT('"state_change_time": "',State_chage_time),'",');
_arrTemp[3]:='"data": {';
_sData[0]:=F_Join_L(ADR(_arrTemp),SIZEOF(_arrTemp[0]),3,ADR(''),SIZEOF(''));
_sData[1]:=M_GetData(arrDataName,arrDataValue,iDataCount);
_sData[2]:='}}';
M_State:=F_Join_L(ADR(_sData),SIZEOF(_sData[0]),2,ADR(''),SIZEOF(''));
END_METHOD

END_PROGRAM

// Http/POUs/FB_HttpClient1
FUNCTION_BLOCK FB_HttpClient1
VAR_INPUT
	Execute:						BOOL;
	Uri:							STRING;
	HostName:						STRING;// Ip
	HostPort:						UINT;// Port
	SendData:						PVOID;
	SendDataLen:					UINT;
	ReceiveData:					PVOID;
	ReceiveDataLen:					UINT;
	Command:						E_HttpRequestOrder:=E_HttpRequestOrder.POST;
END_VAR
VAR_OUTPUT
	Done:							BOOL;
	Busy:							BOOL;
	Error:							BOOL;
END_VAR
VAR
	_fbIotHttpClient:					FB_IotHttpClient();
	_fbIotHttpRequest:					FB_IotHttpRequest();
	_fbIotHttpHeaderFieldMap:			FB_IotHttpHeaderFieldMap();
	_run:								INT;
	_i:									INT;
END_VAR

_fbIotHttpClient.sHostName:=HostName;
_fbIotHttpClient.nHostPort:=HostPort;
//_fbIotHttpRequest.sContentType:='application/x-www-form-urlencoded';
_fbIotHttpClient.Execute();
A_Run();

ACTION A_Run:
{attribute'hide'}
CASE _run OF
	0:
		Busy:=Done:=FALSE;
		IF Command<>E_HttpRequestOrder.None AND  Execute THEN
			_run:=100;
		END_IF;
	100:
		Error:=FALSE;
		Busy:=TRUE;
		CASE Command  OF
			E_HttpRequestOrder.GET:
				IF SendRequest(ETcIotHttpRequestType.HTTP_GET) THEN
					_run:=1000;
				END_IF
			E_HttpRequestOrder.POST:
				IF SendRequest(ETcIotHttpRequestType.HTTP_POST) THEN
					_run:=1000;
				END_IF
		END_CASE
	1000:
		IF NOT _fbIotHttpRequest.bBusy THEN
			_run:=1100;
		END_IF
	1100:
		IF _fbIotHttpRequest.bError THEN
			Error:=TRUE;
		END_IF
		IF _fbIotHttpRequest.nContentSize<>0 THEN
			_fbIotHttpRequest.GetContent(ReceiveData,ReceiveDataLen,TRUE);
		END_IF;
		_run:=1200;
	1200:
		Busy:=FALSE;
		Done:=TRUE;
		IF NOT Execute THEN
			Done:=FALSE;
			_run:=0;
		END_IF
END_CASE
END_ACTION

{attribute'hide'}
METHOD SendRequest : BOOL
VAR_INPUT
	 eRequestType : ETcIotHttpRequestType;
END_VAR
SendRequest:= _fbIotHttpRequest.SendRequest(sUri:=Uri,fbClient:=_fbIotHttpClient,eRequestType:=eRequestType,pContent:=SendData,nContentSize:=F_LEN(SendData),fbHeader:=_fbIotHttpHeaderFieldMap);
END_METHOD

END_FUNCTION_BLOCK

// Json/POUs/FB_JsonObjV5
FUNCTION_BLOCK FB_JsonObjV5
VAR_INPUT
	bFileJsonToObj:				BOOL;
	bObjToFileJson:				BOOL;
	sFilePath:					STRING;
	pData: 						PVOID;// 结构体
	nData:						UDINT;// 缓存大小
	sText:						STRING(5000);
END_VAR
VAR_OUTPUT
	Busy:					BOOL;
	Error:					BOOL;
	Done:					BOOL;	
END_VAR
VAR
	// json功能块
	fbJsonRWDT : FB_JsonReadWriteDataType;
	fbJsonW : FB_JsonSaxWriter;
	fbJsonDP : FB_JsonDomParser;
	// 保存出的json字符串
	jsonStr : STRING(255);
	// json键值对地址
	ArrAdr : INT;
	// 键数组
	keyArr : ARRAY[0..999] OF STRING;
	// 值数组
	dataArr : ARRAY[0..999] OF STRING(255);
	// 值数据类型-未启用
	typeArr : ARRAY[0..999] OF STRING;
	
	_run:				UINT;
	FileOpen : Tc2_System.FB_FileOpen;
	FileRead : Tc2_System.FB_FileRead;
	FileWrite : Tc2_System.FB_FileWrite;
	FileClose : Tc2_System.FB_FileClose;
	FileHelper: FB_FileHelper;
END_VAR

(*
* 功能 1 输入键（字符串）-值（任意数据类型）自动载入json
* 功能 2 输入键（字符串）自动返回值（任意数据类型，包括自定义数据类型以及JSON）
* 功能 3 JSON数据重置
* 功能 4 输出JSON字符串
* 功能 5 输入JSON字符串，转化为Json对象（取消）
* 功能 6 输入特定结构体对象，直接转化为Json字符串并返回
* 功能 7 输入JSON字符串，转化为结构体
*)

A_FileJsonObj();

ACTION A_FileJsonObj:
{attribute'hide'}
FileHelper(
	Read:= , 
	WriteAllText:= , 
	AppendAllText:= , 
	FilePath:=sFilePath , 
	Buffer:=ADR(sText) , 
	BufferLen:=SIZEOF(sText) , 
	TimeOut:= , 
	Busy=> , 
	Error=> , 
	Done=> );
IF FileHelper.Error THEN
	Error:=TRUE;
END_IF

CASE _run OF
	0:
		Busy:=Done:=FALSE;
		IF bFileJsonToObj OR bObjToFileJson THEN
			_run:=100;
		END_IF
	100:
		_run:=0;
		Error:=FALSE;
		Busy:=TRUE;
		IF bFileJsonToObj THEN
			sText:='';
			_run:=200;
		END_IF;
		IF bObjToFileJson THEN
			_run:=500;
		END_IF
	200:
		FileHelper.Read:=TRUE;
		IF FileHelper.Done THEN
			_run:=SEL(FileHelper.Error,300,1000);
			FileHelper.Read:=FALSE;
		END_IF
	300:
		M_JsonStrToObj(sText,nData,pData);
		_run:=1000;
	500:
		sText:=M_ObjToJsonStr(nData,pData);	
		_run:=600;
	600:
		FileHelper.WriteAllText:=TRUE;
		IF FileHelper.Done THEN
			_run:=1000;
			FileHelper.WriteAllText:=FALSE;
		END_IF
	1000:
		Busy:=FALSE;
		Done:=TRUE;
		IF NOT  bFileJsonToObj AND  NOT  bObjToFileJson THEN
			Done:=FALSE;
			_run:=0;
		END_IF
END_CASE
END_ACTION

METHOD M_AddKeyValue : BOOL
VAR_INPUT
	key : STRING;// JSON键
 	nData : UDINT;// 值变量长度
 	pData : PVOID;// 值变量起始地址
END_VAR
VAR
	typestr : STRING;// 值变量数据类型
	tempstr : STRING;// 临时字符串变量
	keystr : STRING;// 键临时变量
END_VAR
(*
* 功能 1 输入键（字符串）-值（任意数据类型）自动载入json
*)
// 获得值变量的数据类型
typestr := fbJsonRWDT.GetDatatypeNameByAddress(nData := nData, pData := pData);
// 重置Json缓存
fbJsonW.ResetDocument();
// 添加数据到Json缓存
fbJsonRWDT.AddJsonValueFromSymbol(fbJsonW, typestr, nData, pData);
// 将当前缓存转为字符串
tempstr := fbJsonW.GetDocument();
// 将键转换为键格式
keystr := concat('"', concat(key, '"'));
// 写入数组缓存
keyArr[ArrAdr] := keystr;
dataArr[ArrAdr] := tempstr;
typeArr[ArrAdr] := typestr;
// 地址+1
ArrAdr := ArrAdr + 1;
END_METHOD

METHOD M_GetJsonStr : string(1000)
VAR_INPUT
END_VAR
VAR
	i: INT;
END_VAR
(*
* 功能 4 输出JSON字符串
*)
// 起始大括号
M_GetJsonStr := Tc2_Standard.CONCAT(M_GetJsonStr, '{');
// 遍历数据数组
FOR i := 0 TO ArrAdr - 1 BY 1 DO
	// 第二个元素开始要加上逗号分隔
	IF i > 0 THEN
		M_GetJsonStr := Tc2_Standard.CONCAT(M_GetJsonStr, ',');
	END_IF
	// 拼接键
	M_GetJsonStr := Tc2_Standard.CONCAT(M_GetJsonStr, KeyArr[i]);
	// 冒号分隔
	M_GetJsonStr := Tc2_Standard.CONCAT(M_GetJsonStr, ':');
	// 拼接值
	M_GetJsonStr := Tc2_Standard.CONCAT(M_GetJsonStr, dataArr[i]);
END_FOR
// 末尾大括号
M_GetJsonStr := Tc2_Standard.CONCAT(M_GetJsonStr, '}');
END_METHOD

METHOD M_GetKeyValue : BOOL
VAR_INPUT
	key : STRING;// JSON键
 	nData : UDINT;// 值变量返回长度
 	pData : PVOID;// 值变量返回起始地址
END_VAR
VAR
	typestr : STRING;// 值变量数据类型
	i : INT;// 键值
	sJson : string(255);
END_VAR
(*
* 功能 2 输入键（字符串）自动返回值（任意数据类型，包括自定义数据类型以及JSON）
*)
// Json中是否存在数据
IF arradr > 0 THEN
	// 获得值变量的数据类型
	typestr := fbJsonRWDT.GetDatatypeNameByAddress(nData := nData, pData := pData);
	// 遍历查找键值
	FOR i := 0 TO ArrAdr - 1 BY 1 DO
		// 给key拼接上""，判断键是否相等
		IF keyarr[i] = concat('"', concat(key, '"')) THEN
			// 如果相等，则返回值
			fbJsonRWDT.SetSymbolFromJson(sJson:= dataarr[i], sDatatype:= typestr, nData := nData, pData := pData);
			EXIT;
		END_IF
	END_FOR
END_IF
END_METHOD

METHOD M_JsonStrToObj
VAR_INPUT
	JsonStr: STRING(5000);
	nData: 	UDINT;
	pData: 	PVOID;
END_VAR
VAR
	typestr: STRING;
END_VAR
(*
* 功能 7 输入JSON字符串，转化为结构体
*)
// 获得值变量的数据类型
typestr := fbJsonRWDT.GetDatatypeNameByAddress(nData := nData, pData := pData);
// 重置Json缓存
fbJsonW.ResetDocument();
// 将JSON字符串的信息写入特定数据
fbJsonRWDT.SetSymbolFromJson(sJson:= JsonStr, sDatatype:= typestr, nData:= nData, pData:= pData);
END_METHOD

METHOD M_ObjToJsonStr : STRING(5000);
VAR_INPUT
	nData: UDINT;
	pData: PVOID;
END_VAR
VAR
	typestr: STRING;
END_VAR
(*
* 功能 6 输入特定结构体对象，直接转化为Json字符串并返回
*)
// 获得值变量的数据类型
typestr := fbJsonRWDT.GetDatatypeNameByAddress(nData := nData, pData := pData);
// 重置Json缓存
fbJsonW.ResetDocument();
// 添加数据到Json缓存
fbJsonRWDT.AddJsonValueFromSymbol(fbJsonW, typestr, nData, pData);
// 将当前缓存转为字符串
fbJsonW.CopyDocument(pDoc:= M_ObjToJsonStr, nDoc:= SIZEOF(M_ObjToJsonStr));
END_METHOD

METHOD M_ResetObj : BOOL
VAR_INPUT
END_VAR
(*
* 功能 3 JSON数据重置
*)
// json键值对地址重置为0
ArrAdr := 0;
END_METHOD

END_FUNCTION_BLOCK

// Matrix2D/FB_Matrix2D
FUNCTION_BLOCK FB_Matrix2D
VAR_INPUT
	X_Home:				LREAL;// X轴起始点
	Y_Home:				LREAL;// Y轴起始点
	XCount:				UINT:=1;// X轴坐标点位数量 从1开始
	XInterval:			LREAL;// X轴间距
	YInterval:			LREAL;// Y轴间距
END_VAR
VAR_OUTPUT
	XPosition:			LREAL;// X轴绝对位置
	YPosition:			LREAL;// Y轴绝对位置
END_VAR
VAR
END_VAR

METHOD M_Index_S : ST_Matrix2DCoordinate
VAR_INPUT
	Index:				UINT;// 位置序号(从0开始)
END_VAR
VAR
	_temp:				DINT;
	_temp1:				DINT;
END_VAR
IF XCount=0 THEN RETURN; END_IF
_temp:=TRUNC(Index/XCount);
_temp1:=Index MOD XCount;
M_Index_S:=SEL((_temp MOD 2)<>0,M_Index_Z(Index),M_XY(XCount-_temp1-1,_temp));
END_METHOD

METHOD M_Index_Z : ST_Matrix2DCoordinate
VAR_INPUT
	Index:				UINT;// 位置序号(从0开始)
END_VAR
VAR
END_VAR
IF XCount=0 THEN RETURN; END_IF
M_Index_Z:=M_XY(Index MOD XCount,TRUNC(Index/XCount));
END_METHOD

METHOD M_XY : ST_Matrix2DCoordinate
VAR_INPUT
	X:					DINT;// 从0开始
	Y:					DINT;// 从0开始
END_VAR
IF XCount=0 THEN RETURN; END_IF

XPosition:= M_XY.X:=X*XInterval+X_Home;
YPosition:=M_XY.Y:=Y*YInterval+Y_Home;
END_METHOD

END_FUNCTION_BLOCK

// ModbusTcp/FB_ModbusTcpClient
FUNCTION_BLOCK FB_ModbusTcpClient
VAR_INPUT
	IP:							STRING;// IP地址
	Port:						UINT:=502;// IP端口号
	UnitID:						BYTE:=11;// MODBUS端口号(自定义)
	Execute:					BOOL;
	TimeOut:					TIME:=T#3S;
	Commend:					E_ModbusClientTcpCmd;
	nMBAddr:					WORD;// 读写起始地址
	nQuantity:					WORD;// 读写数量
	pDestAddr:					PVOID;// 读写数据区
	cbLength:					UINT;// 读写数据区大小
END_VAR
VAR_OUTPUT
	Busy:						BOOL;
	Error:						BOOL;
	Done:						BOOL;
END_VAR
VAR
	_fbMBReadRegs:				FB_MBReadRegs;
	_fbMBReadCoils:				FB_MBReadCoils;
	_fbMBWriteRegs:				FB_MBWriteRegs;
	_fbMBWriteCoils:			FB_MBWriteCoils;
	_iRun:						UINT;
	_busy:						BOOL;
	_ton:						TON;
END_VAR

_fbMBReadCoils(
	sIPAddr:=IP , 
	nTCPPort:=Port , 
	nUnitID:= UnitID, 
	nQuantity:=nQuantity , 
	nMBAddr:=nMBAddr , 
	cbLength:=cbLength , 
	pDestAddr:=pDestAddr , 
	bExecute:= , 
	tTimeout:= , 
	bBusy=> , 
	bError=> , 
	nErrId=> , 
	cbRead=> );
	
_fbMBReadRegs(
	sIPAddr:=IP , 
	nTCPPort:=Port , 
	nUnitID:=UnitID , 
	nQuantity:=nQuantity , 
	nMBAddr:=nMBAddr , 
	cbLength:=cbLength , 
	pDestAddr:=pDestAddr , 
	bExecute:= , 
	tTimeout:= , 
	bBusy=> , 
	bError=> , 
	nErrId=> , 
	cbRead=> );
	
_fbMBWriteRegs(
	sIPAddr:=IP , 
	nTCPPort:=Port , 
	nUnitID:=UnitID , 
	nQuantity:=nQuantity , 
	nMBAddr:=nMBAddr , 
	cbLength:=cbLength, 
	pSrcAddr:=pDestAddr , 
	bExecute:= , 
	tTimeout:= , 
	bBusy=> , 
	bError=> , 
	nErrId=> );
	
_fbMBWriteCoils(
	sIPAddr:=IP , 
	nTCPPort:=Port , 
	nUnitID:=UnitID , 
	nQuantity:=nQuantity , 
	nMBAddr:=nMBAddr , 
	cbLength:=cbLength , 
	pSrcAddr:=pDestAddr , 
	bExecute:= , 
	tTimeout:= , 
	bBusy=> , 
	bError=> , 
	nErrId=> );
	
A_Run();

	
_ton(IN:=Busy , PT:=TimeOut , Q=> , ET=> );

ACTION A_Run:
{attribute'hide'}

_busy:=_fbMBReadCoils.bBusy OR  _fbMBReadRegs.bBusy OR _fbMBWriteRegs.bBusy OR _fbMBWriteCoils.bBusy ;

IF Commend=E_ModbusClientTcpCmd.Reset AND Execute THEN
	_iRun:=0;
	Error:=FALSE;
END_IF


CASE _iRun OF
	0:
		Done:=Busy:=FALSE;
		_fbMBReadCoils.bExecute:=FALSE;
		_fbMBReadRegs.bExecute:=FALSE;
		_fbMBWriteRegs.bExecute:=FALSE;	
		_fbMBWriteCoils.bExecute:=FALSE;
		IF Commend<>E_ModbusClientTcpCmd.None AND Commend<>E_ModbusClientTcpCmd.Reset AND  Execute THEN
			_iRun:=100;
		END_IF
	100:
		Busy:=TRUE;
		Error:=FALSE;
		CASE Commend OF
			E_ModbusClientTcpCmd.ReadCoils:
				_fbMBReadCoils.bExecute:=TRUE;
			E_ModbusClientTcpCmd.ReadRegs:
				_fbMBReadRegs.bExecute:=TRUE;
			E_ModbusClientTcpCmd.WriteRegs:
				_fbMBWriteRegs.bExecute:=TRUE;	
			E_ModbusClientTcpCmd.WriteCoils:
				_fbMBWriteCoils.bExecute:=TRUE;
			ELSE
				_iRun:=10000;
		END_CASE
		IF _busy THEN
			_iRun:=200;
		END_IF
		IF _ton.Q THEN
			Error:=TRUE;
			_iRun:=10000;
		END_IF
	200:
		IF NOT _busy THEN
			_iRun:=300;
		END_IF
	300:
		CASE Commend OF
			E_ModbusClientTcpCmd.ReadCoils:
				IF _fbMBReadCoils.bError THEN
					Error:=TRUE;
				END_IF
			E_ModbusClientTcpCmd.ReadRegs:
				IF  _fbMBReadRegs.bError THEN
					Error:=TRUE;
				END_IF
			E_ModbusClientTcpCmd.WriteRegs:
				IF _fbMBWriteRegs.bError THEN
					Error:=TRUE;
				END_IF
			E_ModbusClientTcpCmd.WriteCoils:
				IF _fbMBWriteCoils.bError THEN
					Error:=TRUE;
				END_IF
		END_CASE
		_iRun:=10000;
	10000:
		Busy:=FALSE;
		Done:=TRUE;
		IF Execute THEN
			Done:=FALSE;
			_iRun:=0;
		END_IF
END_CASE
END_ACTION

END_FUNCTION_BLOCK

// OpcUa/POUS/FB_OpcUaClient
FUNCTION_BLOCK FB_OpcUaClient
VAR_INPUT
	ServerUrl:				STRING;
	NameSpaceUri:			STRING;// NamespaceIndex获取标识
	NamespaceIndex:			DINT:=-1;// -1:则自动获取 非负值则固定获取
	Command:				E_OpcUaClientCmd;
	Identifier:				STRING;
	pVariable:				PVOID;
	cbData:					UDINT;
END_VAR
VAR_OUTPUT
	Error:					BOOL;
	Busy:					BOOL;
	Done:					BOOL;
END_VAR
VAR
	fbUA_Connect				:UA_Connect;
	fbUA_GetNamespaceIndex		:UA_GetNamespaceIndex;
	fbUA_NodeGetHandle			:UA_NodeGetHandle;
	fbUA_Read					:UA_Read;
	fbUa_Write					:UA_Write;
	fbUA_Disconnect				:UA_Disconnect;
	_iRun:						UINT;
END_VAR

A_Run();



fbUA_Connect.SessionConnectInfo.tConnectTimeout		:= DEFAULT_ADS_TIMEOUT;					//定时器超时默认为一分钟
fbUA_Connect.SessionConnectInfo.sApplicationName		:= '';									//请随便填
fbUA_Connect.SessionConnectInfo.eSecurityMode		:= eUASecurityMsgMode_None;				//不签名，不加密
fbUA_Connect.SessionConnectInfo.eSecurityPolicyUri	:= eUASecurityPolicy_None;				//无加密策略
fbUA_Connect.SessionConnectInfo.eTransportProfileUri	:= eUATransportProfileUri_UATcp;		//UaTcp传输， 默认值为1


fbUA_Connect( //进行连接
		Execute			:= ,
		ServerUrl		:= ServerUrl, //IP地址
		SessionConnectInfo	:= , //一些链接附加信息
		Timeout				:= DEFAULT_ADS_TIMEOUT,	 // 超时设置
		ConnectionHdl		=> ,			 //输出一个链接句柄
		Done				=> ,
		Busy				=> ,
		Error				=> ,
		ErrorID				=> 	);
			
fbUA_GetNamespaceIndex(
			Execute			:= ,
			ConnectionHdl	:= fbUA_Connect.ConnectionHdl,//链接句柄
			NameSpaceUri	:= NameSpaceUri, //PLC名称，获取方式请参考实验手册
			Timeout			:= DEFAULT_ADS_TIMEOUT,//超时设置
			NamespaceIndex	=> , //plc 句柄
			Done			=> ,
			Busy			=> ,
			Error			=> ,
			ErrorID			=> );

fbUA_NodeGetHandle.NodeID.eIdentifierType	:= eUAIdentifierType_String;
fbUA_NodeGetHandle.NodeID.nNamespaceIndex	:=DINT_TO_UINT(SEL(NamespaceIndex=-1,NamespaceIndex,fbUA_GetNamespaceIndex.NamespaceIndex));
fbUA_NodeGetHandle.NodeID.sIdentifier		:= Identifier;		
fbUA_NodeGetHandle(
		Execute			:= ,
		ConnectionHdl	:= fbUA_Connect.ConnectionHdl, //连接句柄
		NodeID			:=,	
		Timeout			:= DEFAULT_ADS_TIMEOUT,	//标准超时
		NodeHdl			=> , //该功能块将输出变量句柄
		Done			=> ,
		Busy			=> ,
		Error			=> ,
		ErrorID			=> );

fbUA_Read(
	Execute				:= ,
	ConnectionHdl		:= fbUA_Connect.ConnectionHdl, //连接句柄
	NodeHdl				:= fbUA_NodeGetHandle.NodeHdl, //变量句柄
	stNodeAddInfo		:= , //附加信息
	pVariable			:= pVariable, //将变量读出后写入的地址，是由caller功能块传入进来的
	cbData				:= cbData, //将变量读出后写入的地址的大小，由caller功能块传入进来
	Timeout				:= DEFAULT_ADS_TIMEOUT,//基础超时
	Done				=> ,
	Busy				=> ,
	Error				=> ,
	ErrorID				=>);
	
fbUa_Write(
	Execute:= , 
	ConnectionHdl:= fbUA_Connect.ConnectionHdl, 
	NodeHdl:=fbUA_NodeGetHandle.NodeHdl , 
	stNodeAddInfo:= , 
	pVariable:= pVariable, 
	cbData:=cbData , 
	Timeout:=DEFAULT_ADS_TIMEOUT , 
	Done=> , 
	Busy=> , 
	Error=> , 
	ErrorID=> );
	
fbUA_Disconnect(
	Execute:= , 
	ConnectionHdl:=fbUA_Connect.ConnectionHdl, 
	Timeout:=DEFAULT_ADS_TIMEOUT , 
	Done=> , 
	Busy=> , 
	Error=> , 
	ErrorID=> );

ACTION A_Run:
{attribute'hide'}

IF Command=E_OpcUaClientCmd.Reset THEN
	_iRun:=0;
	Error:=FALSE;
END_IF

CASE _iRun OF
	0:
		Busy:=Done:=FALSE;
		fbUA_NodeGetHandle.Execute:=FALSE;
		fbUA_GetNamespaceIndex.Execute:=FALSE;
		fbUA_Read.Execute:=FALSE;
		fbUa_Write.Execute:=FALSE;
		fbUA_Connect.Execute:=FALSE;
		fbUA_Disconnect.Execute:=FALSE;
		IF Command<>E_OpcUaClientCmd.None AND  Command<>E_OpcUaClientCmd.Reset THEN
			_iRun:=100;
		END_IF
	100://0:None;1:Read;2:Write;100:Connect;101:Disconnect;
		Error:=FALSE;
		Busy:=TRUE;
		CASE Command OF
			E_OpcUaClientCmd.Read,E_OpcUaClientCmd.Write:
				_iRun:=SEL(NamespaceIndex=-1,1008,1000);
			E_OpcUaClientCmd.Connect:
				_iRun:=3000;
			E_OpcUaClientCmd.Disconnect:
				_iRun:=3500;
			ELSE
				_iRun:=10000;	
		END_CASE
	1000:
		fbUA_GetNamespaceIndex.Execute:=TRUE;
		IF fbUA_GetNamespaceIndex.Busy THEN
			fbUA_GetNamespaceIndex.Execute:=FALSE;
			_iRun:=1005;	
		END_IF
	1005:
		IF NOT fbUA_GetNamespaceIndex.Busy THEN
			_iRun:=1008;
		END_IF
	1008:
		fbUA_NodeGetHandle.Execute:=TRUE;
		IF fbUA_NodeGetHandle.Busy THEN
			fbUA_NodeGetHandle.Execute:=FALSE;
			_iRun:=1010;
		END_IF
	1010:
		IF NOT fbUA_NodeGetHandle.Busy THEN
			_iRun:=1020;
		END_IF
	1020:
		CASE Command OF
			E_OpcUaClientCmd.Read:
				_iRun:=2000;
			E_OpcUaClientCmd.Write:
				_iRun:=2500;
			ELSE
				_iRun:=10000;
		END_CASE
	2000:
		fbUA_Read.Execute:=TRUE;
		IF fbUA_Read.Busy THEN
			fbUA_Read.Execute:=FALSE;
			_iRun:=2010;
		END_IF
	2010:
		IF NOT fbUA_Read.Busy THEN
			_iRun:=10000;
		END_IF
	2500:
		fbUa_Write.Execute:=TRUE;
		IF fbUa_Write.Busy THEN
			fbUa_Write.Execute:=FALSE;
			_iRun:=2510;
		END_IF
	2510:
		IF NOT fbUa_Write.Busy THEN
			_iRun:=10000;
		END_IF
	3000:
		fbUA_Connect.Execute:=TRUE;
		IF fbUA_Connect.Busy THEN
			fbUA_Connect.Execute:=FALSE;
			_iRun:=3010;
		END_IF
	3010:
		IF NOT fbUA_Connect.Busy THEN
			_iRun:=10000;
		END_IF
	3500:
		 fbUA_Disconnect.Execute:=TRUE;
		 IF fbUA_Disconnect.Busy THEN
			  fbUA_Disconnect.Execute:=FALSE;
			 _iRun:=3510;
		 END_IF
	3510:
		IF NOT fbUA_Disconnect.Busy THEN
			_iRun:=10000;
		END_IF
	10000:
		CASE Command OF
			E_OpcUaClientCmd.Connect:
				IF fbUA_Connect.Error THEN
					Error:=TRUE;
				END_IF
			E_OpcUaClientCmd.Disconnect:
				IF fbUA_Disconnect.Error THEN
					Error:=TRUE;
				END_IF
			E_OpcUaClientCmd.Read:
				IF fbUA_Read.Error OR fbUA_NodeGetHandle.Error THEN
					Error:=TRUE;
				END_IF
			E_OpcUaClientCmd.Write:
				IF fbUa_Write.Error OR fbUA_NodeGetHandle.Error THEN
					Error:=TRUE;
				END_IF
		END_CASE
		_iRun:=11000;
	11000:
		Busy:=false;
		Done:=TRUE;
		IF  Command=E_OpcUaClientCmd.None  THEN
			_iRun:=0;
		END_IF
END_CASE
END_ACTION

END_FUNCTION_BLOCK

// Recipe/POUs/P_Recipe
PROGRAM P_Recipe
VAR
	_bRecipeCreate:						BOOL;
	_bRecipeDelete:						BOOL;
	_bRecipeRead:						BOOL;
	_bRecipeWrite:						BOOL;
	_sRecipeName:						STRING:='Data';
	_sRecipeDefinitionName:				STRING:='Recipes';
	_bLock:								BOOL;
	
	_fbRecipeManCommands:  				Recipe_Management.RecipeManCommands;
	_ton:								TON;
END_VAR

IF _bRecipeCreate  THEN
_fbRecipeManCommands.CreateRecipe(RecipeDefinitionName:=_sRecipeDefinitionName , RecipeName:=_sRecipeName );
ELSIF  _bRecipeDelete THEN
_fbRecipeManCommands.DeleteRecipe(RecipeDefinitionName:=_sRecipeDefinitionName , RecipeName:=_sRecipeName );
ELSIF  _bRecipeRead  THEN
_fbRecipeManCommands.LoadAndWriteRecipe(RecipeDefinitionName:=_sRecipeDefinitionName , RecipeName:=_sRecipeName );
ELSIF  _bRecipeWrite  THEN
_fbRecipeManCommands.ReadAndSaveRecipe(RecipeDefinitionName:=_sRecipeDefinitionName , RecipeName:=_sRecipeName );
END_IF

IF _bRecipeCreate OR _bRecipeDelete OR _bRecipeRead OR _bRecipeWrite THEN
	_bLock:=TRUE;
END_IF
IF _ton.Q THEN;
	_bLock:=FALSE;
END_IF

_ton(IN:=_bLock , PT:=T#2S , Q=> , ET=> );

_bRecipeCreate:=_bRecipeDelete:=_bRecipeRead:=_bRecipeWrite:=FALSE;

END_PROGRAM

// Regex/F_FIND
FUNCTION F_FIND : UDINT
VAR_INPUT
	STR1:			POINTER TO BYTE;
	STR2:			POINTER TO BYTE;
END_VAR
VAR
	_i:				LINT;
	_t:				LINT;
	_iSTR2:			UDINT;
END_VAR

_iSTR2:=F_LEN(STR2);

WHILE STR1[_i]<>0 DO
	_t:=SEL(STR1[_i]<>STR2[_t],_t+1,0);
	_i:=_i+1;
	IF _t>=_iSTR2 THEN 
		F_Find:=LINT_TO_UDINT(_i);
		EXIT;
	ELSE
		F_Find:=0;
	END_IF
END_WHILE

END_FUNCTION

// Regex/F_Join
FUNCTION F_Join : STRING(255)
VAR_INPUT
	In:						POINTER TO STRING;// 输入数组
	Count:					INT;// 数组大小
	Separator:				STRING;// 分隔符
END_VAR
VAR
	_i:						LINT;
	_sTemp:					STRING(500);
END_VAR

_sTemp:=In[0];
FOR _i:=1 TO Count BY 1 DO
	_sTemp:=CONCAT(CONCAT(_sTemp,Separator),In[_i]);
END_FOR
F_Join:=_sTemp;

END_FUNCTION

// Regex/F_Join_L1
FUNCTION F_Join_L1 : STRING(2000)
VAR_INPUT
	In:						POINTER TO BYTE;// 拼接字符串数组
	OneLength:				UDINT;//Sizeof(In[0])
	Count:					INT;// 数组长度
	Separator:				POINTER TO BYTE;// 分隔符
	SeparatorLength:		UDINT;//Sizeof(SeparatorLength)
	sData:					POINTER TO BYTE;
	sDataLen:				UDINT;// sizeof(sData)
END_VAR
VAR
	_i:						LINT;// 输入字符串数组循环
	_t:						LINT;// 单个输入字符串循环
	_f:						LINT;// 输出元素索引
	_a:						LINT;// 
END_VAR

FOR _i:=0 TO Count BY 1 DO
	FOR _t:=(_i*OneLength) TO (OneLength-1)+(OneLength*_i) BY 1 DO
		IF _f>=sDataLen-1 THEN RETURN; END_IF;
		IF In[_t]=0 THEN EXIT; END_IF;
		sData[_f]:=In[_t];
		_f:=_f+1;
	END_FOR
	IF _i=Count THEN
		EXIT;
	END_IF
	FOR _a:=0 TO SeparatorLength-1 BY 1 DO
		IF _f>=sDataLen-1 THEN RETURN; END_IF;
		IF Separator[_a]=0 THEN EXIT; END_IF;
		sData[_f]:=Separator[_a];
		_f:=_f+1;
	END_FOR
END_FOR
sData[_f]:=0;

END_FUNCTION

// Regex/F_MID
FUNCTION F_MID : bool
VAR_INPUT
	In:					POINTER TO BYTE;
	InLength:			UDINT;// Sizeof(InLength)
	Q:					POINTER TO BYTE;
	QLength:			UDINT;// Sizeof(Q)
	Start:				INT;
	End:				INT;
END_VAR
VAR
	_i:					LINT;
	_t:					LINT;
END_VAR

FOR _i:=0 TO (QLength-1) BY 1 DO
	Q[_i]:=0;
END_FOR
FOR _i:=Start TO End BY 1 DO
	IF _t>=QLength-2 OR _i>= InLength-2  THEN EXIT; END_IF;
	Q[_t]:=In[_i];
	_t:=_t+1;
END_FOR

END_FUNCTION

// Regex/F_WString_TO_String_UTF8
FUNCTION F_WString_TO_String_UTF8
VAR_INPUT
	In:				POINTER TO WSTRING;
	Q:				POINTER TO STRING;
	Count:			INT;
END_VAR
VAR
	_i:				INT;
END_VAR

FOR _i:=0 TO Count BY 1 DO
	WSTRING_TO_UTF8(Q[_i],In[_i],SIZEOF(In[_i]));
END_FOR

END_FUNCTION

// System/POUs/FB_AutoAgain
FUNCTION_BLOCK FB_AutoAgain
VAR_INPUT
	Enable:					BOOL;
	ID:						BYTE;// ID(生成ErrorCode使用 如无相关需求可忽略)
	Category:				E_ErrorCategory;// 报警类别(生成ErrorCode使用 如无相关需求可忽略)
	InfoIndex:				BYTE;// 从50开始(生成ErrorCode使用 如无相关需求可忽略)
	Again:					BOOL;// 重试
	Next:					BOOL;// 跳过
	System:					REFERENCE TO ST_System;
	Station:				REFERENCE TO ST_SystemStation;
	Error:					REFERENCE TO ST_Error;
	StepNext: 				UINT;// 下一步号
	StepAgain:				UINT;// 重试步号
	Timeout:				TIME:=T#1100H;// 确认延迟
	ErrorMessage:			WSTRING;// 提示文本(中文)
	ErrorPosition:			WSTRING;// 发生位置(中文)
	Language:				ARRAY[0..E_Language.MaxCount] OF WSTRING;
END_VAR
VAR_OUTPUT
	Erroring:				BOOL;
	Againg:					BOOL;
	ErrorCode:				DWORD;
END_VAR
VAR
	_ton:					TON;
	_fbErrorTrg:			FB_ErrorTag;
	_fbPulse:				FB_Pulse;
	_fTRIG:					F_TRIG;
	_iRun:					INT;
	_end:					BOOL;
END_VAR

_ton(IN:=Enable AND System.stMode.stDeviceEnable.bAuto AND NOT _end, PT:=Timeout , Q=> , ET=> );
_fbPulse(PT:=T#0.5S , Q=> );

IF NOT Enable THEN
	_iRun:=0;
END_IF

CASE _iRun OF
	0:
		_end:=Againg:=FALSE;
		IF Enable AND System.stMode.stDeviceEnable.bAuto THEN
			Againg:=TRUE;
		END_IF
		IF  Enable AND Again AND System.stMode.stDeviceEnable.bAuto THEN
			Station.iStepNext:=StepAgain;
			_iRun:=200;
		END_IF
		IF _ton.Q OR Next THEN
			Station.iStepNext:=StepNext;
			_iRun:=200;
		END_IF
	200:
		_end:=TRUE;
		Againg:=FALSE;
		IF NOT Enable THEN
			_end:=FALSE;
			_iRun:=0;
		END_IF
END_CASE

_fbErrorTrg(
	System:=System , 
	Error:=Error , 
	ID:=ID , 
	Category:=Category, 
	InfoIndex:=InfoIndex , 
	Enable:=Enable AND ErrorMessage<>"" , 
	Message:=ErrorMessage , 
	Level:=5 , 
	Position:=ErrorPosition , 
	ErrorTime:= T#100MS, 
	Language:= Language, 
	Erroring=>Erroring , 
	ErrorCode=>ErrorCode );

END_FUNCTION_BLOCK

// System/POUs/FB_Pulse
FUNCTION_BLOCK FB_Pulse
VAR_INPUT
	PT:						TIME;
END_VAR
VAR_OUTPUT
	Q:						BOOL;
END_VAR
VAR
	_ton1:					TON;
	_ton2:					TON;
END_VAR

// 脉冲信号
_ton1(IN:= , PT:= PT, Q=> , ET=> );
_ton2(IN:= , PT:= PT, Q=> , ET=> );

IF NOT Q THEN
	_ton1.IN:=TRUE;
	_ton2.IN:=FALSE;
END_IF;

IF Q THEN
	_ton1.IN:=FALSE;
	_ton2.IN:=TRUE;
END_IF;

IF _ton1.Q THEN
	Q:=TRUE;
END_IF;

IF _ton2.Q THEN
	Q:=FALSE;
END_IF;

END_FUNCTION_BLOCK

// System/POUs/FB_Beacon
FUNCTION_BLOCK FB_Beacon
VAR_INPUT
	System:						REFERENCE TO ST_System;
END_VAR
VAR_INPUT
END_VAR
VAR_OUTPUT
END_VAR
VAR
	_fbPulse:					FB_Pulse;
	_bAlarm123:					BOOL;
END_VAR

// 塔灯
_bAlarm123:=System.stMode.arrAlarm[1] OR System.stMode.arrAlarm[2] OR System.stMode.arrAlarm[3];
// 三色灯
_fbPulse(PT:=T#1S , Q=> );

System.stOutput.bLightRed:=_bAlarm123;// 1-3级报警 红灯常亮

System.stOutput.bLightYellow:=NOT _bAlarm123 AND(System.stMode.bStop OR System.stMode.bManual);// 设备正常停止 黄灯常亮

System.stOutput.bLightGreen:=NOT _bAlarm123 AND (System.stMode.bAutoRunning OR System.stMode.bHoming OR System.stMode.bPause);//设备正常运行 绿灯常亮

IF System.stOutput.bLightGreen AND (System.stMode.arrAlarm[4] OR System.stMode.arrAlarm[5]) THEN// 设备正常运行 但有提示信息 绿灯闪烁
	 System.stOutput.bLightGreen:=_fbPulse.Q;
END_IF;
IF System.stOutput.bLightYellow AND (System.stMode.arrAlarm[4] OR System.stMode.arrAlarm[5]) THEN// 设备正常停止 但有提示信息 黄灯闪烁
	 System.stOutput.bLightYellow:=_fbPulse.Q;
END_IF;

System.stOutput.bBuzzer:=_bAlarm123 AND NOT System.stMode.bManual AND  _fbPulse.Q AND NOT System.stInput.bQuiet;// 1-3级报警 并且 非手动状态 蜂鸣器响

END_FUNCTION_BLOCK

// System/POUs/FB_Bool
FUNCTION_BLOCK FB_Bool
VAR_INPUT
	
END_VAR
VAR_OUTPUT
END_VAR
VAR
	_ton:					TON;
	_rTRIG:					R_TRIG;
	_fTRIG:					F_TRIG;
END_VAR

_fTRIG(CLK:= , Q=> );
_rTRIG(CLK:= , Q=> );
_ton(IN:= , PT:= , Q=> , ET=> );

METHOD M_F_TRIG : BOOL
VAR_INPUT
	In:						BOOL;
END_VAR
M_F_TRIG:=_fTRIG.Q;
END_METHOD

METHOD M_R_TRIG : BOOL
VAR_INPUT
	In:						BOOL;
END_VAR
M_R_TRIG:=_rTRIG.Q;
END_METHOD

METHOD M_TON : BOOL
VAR_INPUT
	In:							BOOL;
	Te:							TIME;
END_VAR
_ton.PT:=Te;
_ton.IN:=In;
M_TON:=_ton.Q;
END_METHOD

END_FUNCTION_BLOCK

// System/POUs/FB_Button
FUNCTION_BLOCK FB_Button
VAR_INPUT
	In:				REFERENCE TO BOOL;// 状态写入
	CLK:			BOOL;// 采集de边缘信号
END_VAR
VAR_OUTPUT
END_VAR
VAR
	_rTRIG:				R_TRIG;
	_fTRIG:				F_TRIG;
END_VAR

_rTRIG(CLK:=CLK , Q=> );
_fTRIG(CLK:=CLK , Q=> );

IF _rTRIG.Q THEN
	In:=TRUE;
END_IF

IF _fTRIG.Q THEN
	In:=FALSE;
END_IF

END_FUNCTION_BLOCK

// System/POUs/FB_Memory1
FUNCTION_BLOCK FB_Memory1
VAR_INPUT
	ID:					BYTE;
	Category:			E_ErrorCategory;
	InfoIndex:			BYTE;
	Enable:				BOOL;
	Value:				STRING;// 需要记忆的值
	System:				REFERENCE TO ST_System;
	Error:				REFERENCE TO ST_Error;
	Message:			WSTRING;// 提示信息(中文)
	Position:			WSTRING;// 实例位置
	Language:			ARRAY[0..E_Language.MaxCount] OF WSTRING;
END_VAR
VAR_OUTPUT
	Erroring:			BOOL;
	MemoryValue:		STRING;
END_VAR
VAR
	_iRun:				INT;
	_fbErrorTag:		FB_ErrorTag;
	_ton:				TON;
	_i:					INT;
END_VAR

_ton(IN:=Enable , PT:= T#1S, Q=> , ET=> );
IF NOT _ton.Q  THEN
	MemoryValue:=Value;
END_IF;

_fbErrorTag(
	Error:=Error , 
	System:=System , 
	Enable:= , 
	Message:= , 
	Level:=5 , 
	Position:=Position , 
	ErrorTime:= ,
	Language:=, 
	Erroring=>Erroring,
	ID:=ID,
	Category:=Category,
	InfoIndex:=InfoIndex );


CASE _iRun OF
	0:
		_fbErrorTag.Enable:=FALSE;
		IF MemoryValue<>Value AND _ton.Q THEN
			_iRun:=50;
		END_IF;
	50:
		FOR _i:=0 TO E_Language.MaxCount BY 1 DO
			_fbErrorTag.Language[_i]:=WCONCAT(WCONCAT(Language[_i]," "),TO_WSTRING(MemoryValue));
		END_FOR 
		_iRun:=100;
	100:
		_fbErrorTag.Enable:=TRUE;
		System.stMode.iMemory:=System.stMode.iMemory+1;
		_iRun:=200;
	200:
		IF MemoryValue=Value THEN
			_iRun:=300;
		END_IF;
	300:
		System.stMode.iMemory:=System.stMode.iMemory-1;
		_iRun:=0;
END_CASE;

END_FUNCTION_BLOCK

// System/POUs/FB_System
FUNCTION_BLOCK FB_System
VAR_INPUT
	System:						REFERENCE TO ST_System;
	Error:						REFERENCE TO ST_Error;
	Station:					POINTER TO ST_SystemStation;// 工站
	StationCount:				INT;// 工站数量(从1开始)
END_VAR
VAR_OUTPUT
END_VAR
VAR// SystemDate
	_fbLocalSystemTime:			FB_LocalSystemTime;
	_sYear:						STRING;
	_sMonth:					STRING;
	_sDay:						STRING;
	_sHour:						STRING;
	_sMinute:					STRING;
	_sSecond:					STRING;
	_sMilliseconds:				STRING;
END_VAR
VAR
	_i:							INT;
	_t:							INT;
	_bTransferDone:				BOOL;
	_iAutoModeRun:				INT;
	_sTemp:						WSTRING;
	_bIdle:						BOOL;
	_Idle_Ton:					TON;
	_iInitRun:					INT;
	_iCount:					INT;
	_ton:						ARRAY[0..10] OF TON;
	
	_fbLog:						FB_LogHelper_B;
	
	_fbBeacon:					FB_Beacon;
	
	
	_stNullInfo:				ST_ErrorInfo;
	_arrLogTemp:				ARRAY[0..5] OF STRING;
	_sFifoWrite:				WSTRING(255);
	_fbLogError:				FB_LogHelper_B;
END_VAR

A_Log();// 日志

A_ModeEtop();// 急停状态

A_ModeNone();// 空状态

A_ModeMemory();// 记忆

A_ModeAlarm();// 报警状态

A_ModeAuto();// 自动状态

A_ModeManual();// 手动状态

A_ModeStop();//停止状态

A_ModePause();// 暂停状态

A_ModeHomeDone();// 初始化完成

A_ModeHoming();// 初始化中

A_ModeAutoRunning();// 自动运行

A_ModeBreakpoint();// 断点模式

A_SystemDate();// 获取系统时间

A_ModeDevice();// 元器件执行状态

A_ModeSetting();// 设置模式

A_NowMode();// 当前设备模式显示

A_StepAlternate();// 步数交替

A_ModeInit();// 初始化简化流程


_fbBeacon(System:=System );// 塔灯

ACTION A_Log:
{attribute'hide'}

_fbLog(System:=System , 
		FliePath:=System.stLogConfig.sFilePath , 
		Message:= );
END_ACTION

ACTION A_ModeAlarm:
{attribute'hide'}

IF System.stInput.bReset OR System.stInput.bResetAlarm THEN
	FOR _i:=1 TO 5 BY 1 DO// 清除1-5级报警
		System.stMode.arrAlarm[_i]:=FALSE;
	END_FOR;
	
	FOR _i:=0 TO 100 BY 1 DO// 清除单工站报警
		System.stMode.arrAlarmStation[_i]:=FALSE;
	END_FOR;
END_IF;

System.stMode.bAlarming:=FALSE;
FOR _i:=1 TO 5 BY 1 DO// 1-5级报警
	IF System.stMode.arrAlarm[_i] THEN
		System.stMode.bAlarming:=TRUE;
		EXIT;
	END_IF;
END_FOR;
FOR _i:=0 TO 100 BY 1 DO// 单工站报警
	IF System.stMode.arrAlarmStation[_i] THEN
		System.stMode.bAlarming:=TRUE;
		EXIT;
	END_IF;
END_FOR;




IF System.stInput.bReset OR System.stInput.bResetAlarm THEN
	FOR _i:=0 TO Error.stNow.iCount BY 1 DO
		Error.stNow.arrInfo[_i]:=_stNullInfo;
	END_FOR
END_IF

_fbLogError(System:=System , FliePath:=Error.sFileLogPath , Message:= );

FOR _i:=0 TO Error.stHistory.iCount BY 1 DO
	IF Error.stHistory.arrInfo[_i].bStatus AND Error.bSaveLog THEN
		_arrLogTemp[0]:=Error.stHistory.arrInfo[_i].sSystemDate;
		_arrLogTemp[1]:=Error.stHistory.arrInfo[_i].sLevel;
		_sFifoWrite:=STRING_TO_WSTRING(F_Join(ADR(_arrLogTemp),1,','));
		_fbLogError.Message:=WCONCAT(WCONCAT(WCONCAT(WCONCAT(_sFifoWrite,","),Error.stHistory.arrInfo[_i].sPosition),","),Error.stHistory.arrInfo[_i].arrMessage[Error.eLanguage]);
		_fbLogError.A_AddTail();
		Error.stHistory.arrInfo[_i].bStatus:=FALSE;
	END_IF
END_FOR

GVL.FbErrorLog(
	Read:= , 
	WriteAllText:= , 
	AppendAllText:= , 
	FilePath:='C:\TwinCAT\Error.txt' , 
	Buffer:=ADR(GVL.sErrorInfo) , 
	BufferLen:=SIZEOF(GVL.sErrorInfo) , 
	TimeOut:= , 
	Busy=> , 
	Error=> , 
	Done=> );
END_ACTION

ACTION A_ModeAuto:
{attribute'hide'}

IF System.stMode.bNone AND System.stInput.bAuto  THEN
	System.stMode.bAuto:=TRUE;
END_IF;
IF System.stMode.bEStop OR System.stInput.bReset OR System.stMode.arrAlarm[1] THEN
	System.stMode.bAuto:=FALSE;
END_IF;
END_ACTION

ACTION A_ModeAutoRunning:
{attribute'hide'}

IF System.stMode.bAuto AND System.stMode.bHomeDone AND NOT System.stMode.bStop AND NOT System.stMode.bPause  THEN
	IF System.stInput.bStart  THEN
		System.stMode.bAutoRunning:=TRUE;
	END_IF;
ELSE
	System.stMode.bAutoRunning:=FALSE;
END_IF;
IF System.stInput.bReset  THEN
	System.stMode.bAutoRunning:=FALSE;
END_IF;
END_ACTION

ACTION A_ModeBreakpoint:
{attribute'hide'}

IF System.stInput.bReset THEN
	System.stMode.bBreakpoint:=FALSE;
END_IF
END_ACTION

ACTION A_ModeDevice:
{attribute'hide'}

// 自动允许执行标志
System.stMode.stDeviceEnable.bAuto:=System.stMode.bAuto AND (System.stMode.bAutoRunning OR System.stMode.bHoming OR System.stMode.bPause);

// 自动复位标志
System.stMode.stDeviceRest.bAuto:=TRUE;
FOR _i:=0 TO StationCount-1 BY 1 DO
	IF Station[_i].iStepNow<>0 THEN
		System.stMode.stDeviceRest.bAuto:=FALSE;
		EXIT;
	END_IF;
END_FOR;
IF NOT System.stMode.bAuto THEN
	System.stMode.stDeviceRest.bAuto:=TRUE;
END_IF;

// 手动允许执行标志
System.stMode.stDeviceEnable.bManual:=System.stMode.bManual OR (System.stMode.bAuto AND System.stMode.bStop AND System.iSafetyLevel=5);

// 手动复位标志
System.stMode.stDeviceRest.bManual:=NOT System.stMode.stDeviceEnable.bManual;
END_ACTION

ACTION A_ModeEtop:
{attribute'hide'}

// 急停状态
IF System.stInput.bEStop THEN
	System.stMode.bEStop:=TRUE;
END_IF;
IF System.stInput.bReset AND NOT System.stInput.bEStop THEN
	System.stMode.bEStop:=FALSE;
END_IF;
END_ACTION

ACTION A_ModeHomeDone:
{attribute'hide'}

System.stMode.bHomeDone:=TRUE;
FOR _i:=0 TO StationCount-1 BY 1 DO
	IF Station[_i].iStepNow<1000 THEN
		System.stMode.bHomeDone:=FALSE;
		EXIT;
	END_IF;
END_FOR;

IF NOT System.stMode.bAuto OR System.stInput.bReset THEN
	System.stMode.bHomeDone:=FALSE;
END_IF;
END_ACTION

ACTION A_ModeHoming:
{attribute'hide'}

IF System.stMode.bAuto AND NOT System.stMode.bHomeDone AND NOT System.stMode.bStop AND NOT System.stMode.bPause  THEN
	IF  System.stInput.bStart  THEN
		System.stMode.bHoming:=TRUE;
	END_IF;
ELSE;
	System.stMode.bHoming:=FALSE;
END_IF;
IF System.stInput.bReset THEN
	System.stMode.bHoming:=FALSE;
END_IF;
END_ACTION

ACTION A_ModeInit:
{attribute'hide'}
_ton[0](IN:=_iInitRun<>0 AND NOT System.stInput.bInit, PT:=T#1S , Q=> , ET=> );
IF _ton[0].Q THEN
	_iInitRun:=0;
	System.stInput.bReset:=FALSE;
	System.stInput.bAuto:=FALSE;
	System.stInput.bStart:=FALSE;
END_IF;

CASE _iInitRun OF
	0:
		_iCount:=0;
		IF System.stInput.bInit THEN
			_iInitRun:=100;
		END_IF;
	100:
		System.stInput.bReset:=TRUE;
		IF NOT System.stMode.bAuto AND NOT System.stMode.bManual AND NOT System.stMode.bSetting THEN
			_iInitRun:=150;
		END_IF;
	150:
		_iCount:=_iCount+1;
		IF _iCount>=5 THEN
			_iInitRun:=200;
		END_IF;
	200:
		_iCount:=0;
		System.stInput.bReset:=FALSE;
		IF System.stMode.bEStop THEN
			_iInitRun:=0;
		ELSE
			_iInitRun:=300;
		END_IF;
	300:
		System.stInput.bAuto:=TRUE;
		IF System.stMode.bAuto THEN
			System.stInput.bAuto:=FALSE;
			_iInitRun:=350;
		END_IF;
	350:
		IF System.stMode.arrAlarm[1] OR System.stMode.arrAlarm[2] OR System.stMode.arrAlarm[3] THEN
			_iInitRun:=0;
		ELSE
			_iInitRun:=400;
		END_IF;
	400:
		System.stInput.bStart:=TRUE;
		IF System.stMode.bHoming OR System.stMode.bAutoRunning THEN
			System.stInput.bStart:=FALSE;
			_iInitRun:=500;
		END_IF;
	500:
		IF NOT System.stInput.bInit THEN
			_iInitRun:=0;
		END_IF;
END_CASE;
END_ACTION

ACTION A_ModeManual:
{attribute'hide'}
IF System.stMode.bNone AND System.stInput.bManual THEN
	System.stMode.bManual:=TRUE;
END_IF;
IF System.stMode.bEStop OR System.stInput.bReset THEN
	System.stMode.bManual:=FALSE;
END_IF;
END_ACTION

ACTION A_ModeMemory:
{attribute'hide'}
IF System.stInput.bReset OR NOT System.stMode.bAuto OR NOT System.stMode.bStop THEN
	System.stMode.iMemory:=0;
END_IF;
END_ACTION

ACTION A_ModeNone:
{attribute'hide'}
System.stMode.bNone:= NOT System.stMode.bAuto AND NOT System.stMode.bEStop AND NOT System.stMode.bManual AND NOT System.stMode.bSetting ;
END_ACTION

ACTION A_ModePause:
{attribute'hide'}

IF System.stMode.bAuto AND NOT System.stMode.bStop  THEN
	IF System.stInput.bPause THEN
		System.stMode.bPause:=TRUE;
	ELSIF System.stInput.bStart THEN
		System.stMode.bPause:=FALSE;
	END_IF;
END_IF;
IF NOT System.stMode.bAuto OR System.stMode.bStop OR System.stInput.bReset THEN
	System.stMode.bPause:=FALSE;
END_IF;
END_ACTION

ACTION A_ModeSetting:
{attribute'hide'}
IF System.stMode.bNone AND System.stInput.bSetting THEN
	System.stMode.bSetting:=TRUE;
END_IF;
IF System.stInput.bReset OR System.stMode.bEStop THEN
	System.stMode.bSetting:=FALSE;
END_IF;
END_ACTION

ACTION A_ModeStop:
{attribute'hide'}
IF System.stMode.bAuto THEN
	IF System.stMode.arrAlarm[1] OR System.stMode.arrAlarm[2] OR System.stMode.arrAlarm[3] OR System.stInput.bStop THEN
		System.stMode.bStop:=TRUE;
	ELSIF System.stInput.bStart  AND System.stMode.iMemory=0 THEN
		System.stMode.bStop:=FALSE;
	END_IF;
END_IF;
IF NOT System.stMode.bAuto OR System.stInput.bReset THEN
	System.stMode.bStop:=FALSE;
END_IF;
END_ACTION

ACTION A_NowMode:
{attribute'hide'}
System.stMode.sNowMode:='None';
IF System.stMode.bAuto THEN
	System.stMode.sNowMode:='Auto';
END_IF;
IF System.stMode.bHomeDone THEN
	System.stMode.sNowMode:='HomeDone';
END_IF;
IF System.stMode.bHoming THEN
	System.stMode.sNowMode:='Homing';
END_IF;
IF System.stMode.bAutoRunning THEN
	System.stMode.sNowMode:='AutoRunning';
END_IF;
IF System.stMode.bIdle THEN
	System.stMode.sNowMode:='Idle';
END_IF;
IF System.stMode.bPause THEN
	System.stMode.sNowMode:='Pause';
END_IF;
IF System.stMode.bStop THEN
	System.stMode.sNowMode:='Stop';
END_IF;
IF System.stMode.bAlarming THEN
	System.stMode.sNowMode:='Alarm';
END_IF;
IF System.stMode.bManual THEN
	System.stMode.sNowMode:='Manual';
END_IF;
IF System.stMode.bSetting THEN
	System.stMode.sNowMode:='Setting';
END_IF;
IF System.stMode.bEStop THEN
	System.stMode.sNowMode:='EStop';
END_IF;
END_ACTION

ACTION A_StepAlternate:
{attribute'hide'}
_bIdle:=TRUE;// 空闲状态
FOR _i:=0 TO StationCount-1 BY 1 DO	
	// 步数传递
	IF (System.stMode.bHoming AND Station[_i].iStepNow<1000) OR // 初始化中
		(System.stMode.bAutoRunning AND Station[_i].iStepNow>=1000) OR// 自动运行 
		(System.stMode.bPause AND (Station[_i].iStepNow MOD 10)<>0) THEN// 暂停
		
		IF Station[_i].iStepNow<>Station[_i].iStepNext AND NOT System.stMode.arrAlarmStation[_i]  THEN
			IF NOT System.stMode.bBreakpoint OR (System.stMode.bBreakpoint AND System.stInput.bStart) THEN
				
				// 用于保存历史步
				FOR _t:=9 TO 1 BY -1 DO
					Station[_i].arrStepHistory[_t]:=Station[_i].arrStepHistory[_t-1];
				END_FOR;
				Station[_i].arrStepHistory[0].iStep:=Station[_i].iStepPrev:=Station[_i].iStepNow;
				Station[_i].arrStepHistory[0].arrInfo:=Station[_i].arrInfo;
				Station[_i].arrStepHistory[0].arrName:=Station[_i].arrName;
			
				// 保存日志
				IF System.stLogConfig.bExecute THEN
					_fbLog.Message:=WCONCAT(WCONCAT( WCONCAT( WCONCAT(WCONCAT(WCONCAT(TO_WSTRING(System.stSystemDate.sNow),","),Station[_i].arrName[System.stLogConfig.eLanguage]),","),TO_WSTRING(Station[_i].iStepNow)),","),Station[_i].arrInfo[System.stLogConfig.eLanguage]);
					_fbLog.A_AddTail();
				END_IF;

				// 用于传递当前步
				Station[_i].iStepNow:=Station[_i].iStepNext;
			
				// 空闲状态
				_bIdle:=FALSE;	
				
			END_IF
		END_IF;
	END_IF;
END_FOR;

_Idle_Ton(IN:=_bIdle AND System.stMode.bAutoRunning , PT:=T#60S , Q=>System.stMode.bIdle , ET=> );

IF System.stMode.bEStop OR System.stMode.arrAlarm[1] OR System.stMode.arrAlarm[2] OR NOT System.stMode.bAuto THEN
	FOR _i:=0 TO StationCount-1 BY 1 DO
		Station[_i].iStepPrev:=0;
		Station[_i].iStepNext:=0;
		Station[_i].iStepNow:=0;
	END_FOR;
END_IF;
END_ACTION

ACTION A_SystemDate:
{attribute'hide'}
_fbLocalSystemTime(
	sNetID:= , 
	bEnable:=TRUE , 
	dwCycle:= , 
	dwOpt:= , 
	tTimeout:= , 
	bValid=> , 
	systemTime=> , 
	tzID=> );

System.stSystemDate.iYear:=WORD_TO_INT(_fbLocalSystemTime.SystemTIME.wYear);
System.stSystemDate.iMonth:=WORD_TO_INT(_fbLocalSystemTime.SystemTIME.wMonth);
System.stSystemDate.iDay:=WORD_TO_INT(_fbLocalSystemTime.SystemTIME.wDay);
System.stSystemDate.iHour:=WORD_TO_INT(_fbLocalSystemTime.SystemTIME.wHour);
System.stSystemDate.iMinute:=WORD_TO_INT(_fbLocalSystemTime.SystemTIME.wMinute);
System.stSystemDate.iSecond:=WORD_TO_INT(_fbLocalSystemTime.SystemTIME.wSecond);
System.stSystemDate.iMilliseconds:=WORD_TO_INT(_fbLocalSystemTime.SystemTIME.wMilliseconds);

System.stSystemDate.sDateDay:=CONCAT(CONCAT(CONCAT(CONCAT(TO_STRING(System.stSystemDate.iYear),'-'),M_Join0(System.stSystemDate.iMonth)),'-'),M_Join0(System.stSystemDate.iDay));

// 获取系统时间
_sDay:= CONCAT((System.stSystemDate.sDateDay),' ');
_sHour:= CONCAT(M_Join0(System.stSystemDate.iHour),'.');
_sMinute:= CONCAT(M_join0(System.stSystemDate.iMinute),'.');
_sSecond:= CONCAT(M_join0(System.stSystemDate.iSecond),'.');
_sMilliseconds:=INT_TO_STRING(System.stSystemDate.iMilliseconds);

System.stSystemDate.sNow:=CONCAT(CONCAT(CONCAT(CONCAT(CONCAT(CONCAT(_sYear,_sMonth),_sDay),_sHour),_sMinute),_sSecond),_sMilliseconds);
END_ACTION

END_FUNCTION_BLOCK

// TcpIp/POUs/FB_TcpIpClient
FUNCTION_BLOCK FB_TcpIpClient
VAR_INPUT
	TcpIpClient:					REFERENCE TO ST_TcpIpClient;
	Data:							REFERENCE TO ST_TcpIpData;
	Error:							REFERENCE TO ST_Error;
	System:							REFERENCE TO ST_System;
END_VAR
VAR_OUTPUT
END_VAR
VAR
	_fbSocketConnect:				FB_SocketConnect;
	_fbSocketSend:					FB_SocketSend;
	_fbSocketReceive:				FB_SocketReceive;
	_fbSockClose:					FB_SocketClose;
	_arrFbErrorTag:					ARRAY[0..3] OF FB_ErrorTag;
	_bFistRun:						BOOL:=TRUE;
END_VAR
VAR
	_iSendRun:						INT;
	_iReceiveRun:					INT;
	_arrF:							ARRAY[0..6] OF F_TRIG;
	_arrT:							ARRAY[0..3] OF R_TRIG;	
	_i:								INT;
END_VAR

TcpIpClient.sName:=TcpIpClient.arrInfo[System.stMode.eLanguage].sName;

IF _bFistRun THEN
	A_Init();
END_IF

A_Connect();

A_ControlReset();

A_Receive();

A_Send();

A_Close();

A_Error();

A_Status();

_bFistRun:=FALSE;

ACTION A_Close:
{attribute'hide'}
_fbSockClose(
	sSrvNetId:= , 
	hSocket:=_fbSocketConnect.hSocket , 
	bExecute:= , 
	tTimeout:=T#1S , 
	bBusy=> , 
	bError=> , 
	nErrId=> );
	
_fbSockClose.bExecute:= (System.stMode.stDeviceEnable.bAuto AND TcpIpClient.stContorl.stClose.bAuto) OR 
						(System.stMode.stDeviceEnable.bManual AND TcpIpClient.stContorl.stClose.bManual);
END_ACTION

ACTION A_Connect:
{attribute'hide'}
// 连接
_fbSocketConnect(
	sSrvNetId:='', 
	sRemoteHost:=Data.sServerIp , // 服务器Ip地址
	nRemotePort:=Data.iServerPort , 
	bExecute:= , 
	tTimeout:=T#1S , 
	bBusy=>, 
	bError=> , 
	nErrId=> , 
	hSocket=> );

_fbSocketConnect.bExecute:=(System.stMode.stDeviceEnable.bAuto AND TcpIpClient.stContorl.stConnect.bAuto) OR (System.stMode.stDeviceEnable.bManual AND TcpIpClient.stContorl.stConnect.bManual);
END_ACTION

ACTION A_ControlReset:
{attribute'hide'}
IF System.stMode.stDeviceRest.bAuto THEN
	TcpIpClient.stContorl.stClose.bAuto:=FALSE;
	TcpIpClient.stContorl.stConnect.bAuto:=FALSE;
	TcpIpClient.stContorl.stReceive.bAuto:=FALSE;
	TcpIpClient.stContorl.stSend.bAuto:=FALSE;
END_IF;

IF System.stMode.stDeviceRest.bManual THEN
	TcpIpClient.stContorl.stClose.bManual:=FALSE;
	TcpIpClient.stContorl.stConnect.bManual:=FALSE;
	TcpIpClient.stContorl.stReceive.bManual:=FALSE;
	TcpIpClient.stContorl.stSend.bManual:=FALSE;
END_IF;
END_ACTION

ACTION A_Error:
{attribute'hide'}
_arrT[0](CLK:=_fbSocketConnect.bError , Q=> );
_arrFbErrorTag[0](
	Error:=Error , 
	System:=System , 
	Enable:=_arrT[0].Q, 
	Message:= , 
	Level:=4 , 
	ErrorTime:= ,
	Position:=WCONCAT("FB_TcpIpClient:",TcpIpClient.sName),
	Erroring=>TcpIpClient.stStatus.bErrorConnect,
	ID:=TcpIpClient.ID,
	Category:=E_ErrorCategory.TCP_IP,
	InfoIndex:=0 );
IF _arrFbErrorTag[0].Erroring THEN
	FOR _i:=0 TO E_Language.MaxCount BY 1 DO
		_arrFbErrorTag[0].Language[_i]:=WCONCAT(TcpIpClient.sName,WCONCAT(TcpIpClient.arrInfo[_i].sConnectError,UDINT_TO_WSTRING(_fbSocketConnect.nErrId)));
	END_FOR
END_IF


_arrT[1](CLK:=_fbSocketSend.bError , Q=> );	
_arrFbErrorTag[1](
	Error:=Error , 
	System:=System , 
	Enable:=_arrT[1].Q, 
	Message:=WCONCAT(TcpIpClient.sName,WCONCAT("Tcp/Ip发送错误",UDINT_TO_WSTRING(_fbSocketSend.nErrId))) , 
	Level:=4 , 
	ErrorTime:= ,
	Position:=WCONCAT("FB_TcpIpClient:",TcpIpClient.sName),
	Erroring=>TcpIpClient.stStatus.bErrorSend,
	ID:=TcpIpClient.ID,
	Category:=E_ErrorCategory.TCP_IP,
	InfoIndex:=1);
IF _arrFbErrorTag[1].Erroring THEN
	FOR _i:=0 TO E_Language.MaxCount BY 1 DO
		_arrFbErrorTag[1].Language[_i]:=WCONCAT(TcpIpClient.sName,WCONCAT(TcpIpClient.arrInfo[_i].sSendError,UDINT_TO_WSTRING(_fbSocketSend.nErrId)));
	END_FOR
END_IF


	

_arrT[2](CLK:=_fbSocketReceive.bError , Q=> );	
_arrFbErrorTag[2](
	Error:=Error , 
	System:=System , 
	Enable:=_arrT[2].Q, 
	Message:=WCONCAT(TcpIpClient.sName,WCONCAT("Tcp/Ip接收错误",UDINT_TO_WSTRING(_fbSocketReceive.nErrId))) , 
	Level:=4 , 
	ErrorTime:= ,
	Position:=WCONCAT("FB_TcpIpClient:",TcpIpClient.sName),
	Erroring=>TcpIpClient.stStatus.bErrorReceive,
	ID:=TcpIpClient.ID,
	Category:=E_ErrorCategory.TCP_IP,
	InfoIndex:=2);
IF _arrFbErrorTag[2].Erroring THEN
	FOR _i:=0 TO E_Language.MaxCount BY 1 DO
		_arrFbErrorTag[2].Language[_i]:=WCONCAT(TcpIpClient.sName,WCONCAT(TcpIpClient.arrInfo[_i].sReceiveError,UDINT_TO_WSTRING(_fbSocketReceive.nErrId)));
	END_FOR
END_IF


	

_arrT[3](CLK:=_fbSockClose.bError , Q=> );	
_arrFbErrorTag[3](
	Error:=Error , 
	System:=System , 
	Enable:=_arrT[3].Q, 
	Message:=WCONCAT(TcpIpClient.sName,WCONCAT("Tcp/Ip关闭错误",UDINT_TO_WSTRING(_fbSockClose.nErrId))) , 
	Level:=4 , 
	ErrorTime:=,
	Position:=WCONCAT("FB_TcpIpClient:",TcpIpClient.sName),
	Erroring=>TcpIpClient.stStatus.bErrorClose,
	ID:=TcpIpClient.ID,
	Category:=E_ErrorCategory.TCP_IP,
	InfoIndex:=3);
IF _arrFbErrorTag[3].Erroring THEN
	FOR _i:=0 TO E_Language.MaxCount BY 1 DO
		_arrFbErrorTag[3].Language[_i]:=WCONCAT(TcpIpClient.sName,WCONCAT(TcpIpClient.arrInfo[_i].sCloseError,UDINT_TO_WSTRING(_fbSockClose.nErrId)));
	END_FOR
END_IF
END_ACTION

ACTION A_Init:
{attribute'hide'}
TcpIpClient.arrInfo[E_Language.Chinese].sCloseError:=":Tcp/Ip关闭错误 ";
TcpIpClient.arrInfo[E_Language.Chinese].sConnectError:=":Tcp/Ip连接错误 ";
TcpIpClient.arrInfo[E_Language.Chinese].sReceiveError:=":Tcp/Ip接收错误 ";
TcpIpClient.arrInfo[E_Language.Chinese].sSendError:=":Tcp/Ip发送错误 ";

TcpIpClient.arrInfo[E_Language.English].sCloseError:=":Tcp/Ip Close error ";
TcpIpClient.arrInfo[E_Language.English].sConnectError:=":Tcp/Ip Connect error ";
TcpIpClient.arrInfo[E_Language.English].sReceiveError:=":Tcp/Ip Receive error ";
TcpIpClient.arrInfo[E_Language.English].sSendError:=":Tcp/Ip Send error ";

TcpIpClient.arrInfo[E_Language.Vietnamese].sCloseError:=":Đóng lỗi ";
TcpIpClient.arrInfo[E_Language.Vietnamese].sConnectError:=":Lỗi kết nối ";
TcpIpClient.arrInfo[E_Language.Vietnamese].sReceiveError:=":Nhận lỗi ";
TcpIpClient.arrInfo[E_Language.Vietnamese].sSendError:=":Gửi lỗi ";

TcpIpClient.arrInfo[E_Language.Hindi].sCloseError:=":त्रुटि बंद करें ";
TcpIpClient.arrInfo[E_Language.Hindi].sConnectError:=":एरर कनेक्ट ";
TcpIpClient.arrInfo[E_Language.Hindi].sReceiveError:=":त्रुटि प्राप्त करें ";
TcpIpClient.arrInfo[E_Language.Hindi].sSendError:=":त्रुटि भेजें ";
END_ACTION

ACTION A_Receive:
{attribute'hide'}
_fbSocketReceive.bExecute:=(System.stMode.stDeviceEnable.bAuto AND TcpIpClient.stContorl.stReceive.bAuto) OR (System.stMode.stDeviceEnable.bManual AND TcpIpClient.stContorl.stReceive.bManual);

_arrF[6](CLK:=_fbSocketReceive.bExecute, Q=> );
IF _arrF[6].Q THEN
	TcpIpClient.sReceiveData:='';
END_IF;

// 接收
_fbSocketReceive(
	sSrvNetId:= , 
	hSocket:=_fbSocketConnect.hSocket, 
	cbLen:= SIZEOF(TcpIpClient.sReceiveData), 
	pDest:= ADR(TcpIpClient.sReceiveData), 
	bExecute:= , 
	tTimeout:=T#2S , 
	bBusy=> , 
	bError=> , 
	nErrId=> , 
	nRecBytes=> );
END_ACTION

ACTION A_Send:
{attribute'hide'}
// 发送
_fbSocketSend(
	sSrvNetId:= , 
	hSocket:=_fbSocketConnect.hSocket , // 连接句柄
	cbLen:=F_LEN(ADR(TcpIpClient.sSendData)),
	pSrc:=ADR(TcpIpClient.sSendData) , 
	bExecute:= , 
	tTimeout:=T#2S , 
	bBusy=> , 
	bError=> , 
	nErrId=> );
	
IF (System.stMode.stDeviceEnable.bAuto AND TcpIpClient.stContorl.stSend.bAuto) OR (System.stMode.stDeviceEnable.bManual AND TcpIpClient.stContorl.stSend.bManual) THEN
	_fbSocketSend.bExecute:= TRUE;
ELSE
	_fbSocketSend.bExecute:= FALSE;
END_IF;
END_ACTION

ACTION A_Status:
{attribute'hide'}
TcpIpClient.stStatus.bError:=_fbSocketConnect.bError OR _fbSocketSend.bError OR _fbSocketReceive.bError OR _fbSockClose.bError;

TcpIpClient.stStatus.bConnecting:=_fbSocketConnect.bBusy;
TcpIpClient.stStatus.bReceiving:=_fbSocketReceive.bBusy;
TcpIpClient.stStatus.bSending:=_fbSocketSend.bBusy;
TcpIpClient.stStatus.bClosing:=_fbSockClose.bBusy;

_arrF[0](CLK:=_fbSocketConnect.bBusy , Q=> );
IF _arrF[0].Q AND NOT _fbSocketConnect.bError THEN
	TcpIpClient.stStatus.bConnected:=TRUE;
END_IF;
IF _fbSocketConnect.bBusy OR _fbSocketConnect.bError OR TcpIpClient.stContorl.stClose.bAuto OR TcpIpClient.stContorl.stClose.bManual THEN
	TcpIpClient.stStatus.bConnected:=FALSE;
END_IF;

_arrF[1](CLK:=_fbSocketReceive.bBusy , Q=> );
IF _arrF[1].Q AND  NOT _fbSocketReceive.bError THEN
	TcpIpClient.stStatus.bReceived:=TRUE;
END_IF;
IF _fbSocketReceive.bBusy OR _fbSocketReceive.bError  THEN
	TcpIpClient.stStatus.bReceived:=FALSE;
END_IF;

_arrF[2](CLK:=_fbSocketSend.bBusy , Q=> );
IF _arrF[2].Q AND  NOT _fbSocketSend.bError  THEN
	TcpIpClient.stStatus.bSent:=TRUE;
END_IF;
IF _fbSocketSend.bBusy OR _fbSocketSend.bError  THEN
	TcpIpClient.stStatus.bSent:=FALSE;
END_IF;

_arrF[3](CLK:=_fbSockClose.bBusy , Q=> );
IF _arrF[3].Q AND  NOT _fbSockClose.bError  THEN
	TcpIpClient.stStatus.bClosed:=TRUE;
END_IF;
IF _fbSockClose.bBusy OR _fbSockClose.bError  THEN
	TcpIpClient.stStatus.bClosed:=FALSE;
END_IF;
END_ACTION

END_FUNCTION_BLOCK

// TcpIp/POUs/FB_TcpIpClient1
FUNCTION_BLOCK FB_TcpIpClient1
VAR_INPUT
	IP:					STRING;
	Port:				UINT;
	Command:			E_TcpIpClientCmd;// 触发命令(当收到Done信号后 至None)
	Data:				PVOID;// 读写数据区
	DataLen:			UINT;
END_VAR
VAR_OUTPUT
	Busy:				BOOL;
	Error:				BOOL;
	Done:				BOOL;
END_VAR
VAR
	_fbSocketConnect:				FB_SocketConnect;
	_fbSocketSend:					FB_SocketSend;
	_fbSocketReceive:				FB_SocketReceive;
	_fbSockClose:					FB_SocketClose;
	_run:							UINT;
END_VAR

A_Run();

_fbSocketConnect(
	sSrvNetId:= , 
	sRemoteHost:=IP , 
	nRemotePort:=Port , 
	bExecute:= , 
	tTimeout:= , 
	bBusy=> , 
	bError=> , 
	nErrId=> , 
	hSocket=> );
_fbSocketReceive(
	sSrvNetId:= , 
	hSocket:=_fbSocketConnect.hSocket , 
	cbLen:=DataLen , 
	pDest:=Data , 
	bExecute:= , 
	tTimeout:= , 
	bBusy=> , 
	bError=> , 
	nErrId=> , 
	nRecBytes=> );
_fbSocketSend(
	sSrvNetId:= , 
	hSocket:=_fbSocketConnect.hSocket , 
	cbLen:= DataLen, 
	pSrc:=Data , 
	bExecute:= , 
	tTimeout:= , 
	bBusy=> , 
	bError=> , 
	nErrId=> );
_fbSockClose(
	sSrvNetId:= , 
	hSocket:=_fbSocketConnect.hSocket , 
	bExecute:= , 
	tTimeout:= , 
	bBusy=> , 
	bError=> , 
	nErrId=> );

ACTION A_Run:
{attribute'hide'}
IF Command=E_TcpIpClientCmd.Reset THEN
	_run:=0;
	Error:=FALSE;
END_IF

CASE _run OF
	0:
		Done:=Busy:=FALSE;
		_fbSocketConnect.bExecute:=FALSE;
		_fbSockClose.bExecute:=FALSE;
		_fbSocketReceive.bExecute:=FALSE;
		_fbSocketSend.bExecute:=FALSE;
		IF Command<>E_TcpIpClientCmd.None AND Command<>E_TcpIpClientCmd.Reset THEN
			_run:=100;
		END_IF
	100:
		Error:=FALSE;
		Busy:=TRUE;
		CASE  Command OF
			E_TcpIpClientCmd.Connect:
				_run:=1000;
			E_TcpIpClientCmd.Disconnect:
				_run:=2000;
			E_TcpIpClientCmd.Read:
				_run:=3000;
			E_TcpIpClientCmd.Write:
				_run:=4000;
			ELSE
				_run:=10000;
		END_CASE
	1000:
		_fbSocketConnect.bExecute:=TRUE;
		IF _fbSocketConnect.bBusy THEN
			_fbSocketConnect.bExecute:=FALSE;
			_run:=1100;
		END_IF
	1100:
		IF NOT _fbSocketConnect.bBusy THEN
			_run:=10000;
		END_IF
	2000:
		_fbSockClose.bExecute:=TRUE;
		IF  _fbSockClose.bBusy THEN
			_fbSockClose.bExecute:=FALSE;
			_run:=2100;
		END_IF
	2100:
		IF NOT _fbSockClose.bBusy  THEN
			_run:=10000;
		END_IF
	3000:
		_fbSocketReceive.bExecute:=TRUE;
		IF  _fbSocketReceive.bBusy THEN
			_fbSocketReceive.bExecute:=FALSE;
			_run:=3100;
		END_IF
	3100:
		IF NOT _fbSocketReceive.bBusy THEN
			_run:=10000;
		END_IF
	4000:
		_fbSocketSend.bExecute:=TRUE;
		IF _fbSocketSend.bBusy THEN
			_fbSocketSend.bExecute:=FALSE;
			_run:=4100;
		END_IF
	4100:
		IF NOT  _fbSocketSend.bBusy THEN
			_run:=10000;
		END_IF
	10000:
		CASE  Command OF
			E_TcpIpClientCmd.Connect:
				IF _fbSocketConnect.bError THEN
					Error:=TRUE;
				END_IF
			E_TcpIpClientCmd.Disconnect:
				IF _fbSockClose.bError THEN
					Error:=TRUE;
				END_IF
			E_TcpIpClientCmd.Read:
				IF _fbSocketReceive.bError THEN
					Error:=TRUE;
				END_IF
			E_TcpIpClientCmd.Write:
				IF _fbSocketSend.bError THEN
					Error:=TRUE;
				END_IF
		END_CASE
		_run:=11000;
	11000:
		Busy:=FALSE;
		Done:=TRUE;
		IF Command=E_TcpIpClientCmd.None THEN
			_run:=0;
		END_IF
END_CASE
END_ACTION

END_FUNCTION_BLOCK

// Windows/FB_WindowsCmdAsync
FUNCTION_BLOCK FB_WindowsCmdAsync
VAR_INPUT
	Execute:				BOOL;// 触发使能(在收到Done后 才能False)
	Command:				PVOID;
	FileName:				STRING:='WindowsCmdTempAsync.bat';
END_VAR
VAR_OUTPUT
	Busy:					BOOL;
	Done:					BOOL;
	Error:					BOOL;
END_VAR
VAR
	_fbFielHelper:			FB_FileHelper;
	_StartProcess:			NT_StartProcess;	
	_run:					UINT;
	_path:					STRING;
	_ton:					TON;
END_VAR

_fbFielHelper.FilePath:=_StartProcess.PATHSTR:=CONCAT('C:\TwinCAT\',FileName);

_StartProcess(
	NETID:= , 
	PATHSTR:= , 
	DIRNAME:='C:\TwinCAT\' , 
	COMNDLINE:= , 
	START:= , 
	TMOUT:= , 
	BUSY=> , 
	ERR=> , 
	ERRID=> );
	
_fbFielHelper(
	Read:= , 
	WriteAllText:= , 
	AppendAllText:= , 
	FilePath:= , 
	Buffer:=Command , 
	BufferLen:=F_LEN(Command) , 
	TimeOut:= , 
	Busy=> , 
	Error=> , 
	Done=> );
	
A_Run();

ACTION A_Run:
{attribute'hide'}
IF (_fbFielHelper.Error OR _StartProcess.ERR) AND Done THEN
	Error:=TRUE;
END_IF;

CASE _run OF 
	0:
		_fbFielHelper.WriteAllText:=FALSE;
		_StartProcess.START:=FALSE;
		Busy:=Done:=FALSE;
		IF Execute THEN
			_run:=100;
		END_IF
	100:
		Busy:=TRUE;
		Error:=FALSE;
		_run:=200;
	200:
		_fbFielHelper.WriteAllText:=TRUE;
		IF  _fbFielHelper.Done THEN
			_fbFielHelper.WriteAllText:=FALSE;
			_run:=SEL(_fbFielHelper.Error,300,1000);
		END_IF
	300:
		_StartProcess.START:=TRUE;
		IF _StartProcess.BUSY THEN
			_run:=400;
		END_IF
	400:
		_StartProcess.START:=FALSE;
		IF NOT _StartProcess.BUSY THEN
			_run:=1100;
		END_IF
	1100:
		Busy:=FALSE;
		Done:=TRUE;
		IF NOT Execute THEN
			Done:=FALSE;
			_run:=0;
		END_IF;
END_CASE
END_ACTION

END_FUNCTION_BLOCK

// Yield/POUs/FB_Yield
FUNCTION_BLOCK FB_Yield
VAR_INPUT
	System:			REFERENCE TO ST_System;
	Yield:			REFERENCE TO ST_Yield;
	Data:			REFERENCE TO ST_YieldData;
END_VAR
VAR_OUTPUT
END_VAR
VAR
	_arrR:			ARRAY[0..10] OF	R_TRIG;
	_arrF:			ARRAY[0..10] OF F_TRIG;
	_iAll:			REAL;
	_sTime:			STRING;
	_rTRIG:			R_TRIG;
END_VAR

_sTime:=CONCAT(INT_TO_STRING(System.stSystemDate.iHour),CONCAT(INT_TO_STRING(System.stSystemDate.iMinute),INT_TO_STRING(System.stSystemDate.iSecond)));
_rTRIG(CLK:= ((_sTime='2000')OR (_sTime='800') AND Yield.stControl.bAutoClear), Q=> );
IF System.stInput.bReset THEN
	Yield.stControl.bNG:=FALSE;
	Yield.stControl.bOk:=FALSE;
	Yield.stControl.bTOSS:=FALSE;
END_IF

_arrF[0](CLK:=Yield.stControl.bOk , Q=> );
IF _arrF[0].Q THEN
	Data.iOK:=Data.iOK+1;
END_IF

_arrF[1](CLK:=Yield.stControl.bNG , Q=> );
IF _arrF[1].Q THEN
	Data.iNG:=Data.iNG+1;
END_IF

_arrF[2](CLK:=Yield.stControl.bTOSS , Q=> );
IF _arrF[2].Q THEN
	Data.iTOSS:=Data.iTOSS+1;
END_IF


_iAll:=Data.iAll:=Data.iNG+Data.iOK;


Data.fNgPercentage:=  SEL(Data.iAll=0,Data.iNG/_iAll,0)*100;
Data.fOkPercentage:=SEL(Data.iAll=0,Data.iOK/_iAll,0)*100;
Data.fTOSSPercentage:=SEL((Data.iNG+Data.iOK+Data.iTOSS)=0,Data.iTOSS/(Data.iNG+Data.iOK+Data.iTOSS),0)*100;
IF Yield.stControl.bClear OR _rTRIG.Q THEN
	Data.iOK:=Data.iNG:=Data.iTOSS:=0;
	Data.fNgPercentage:=Data.fOkPercentage:=Data.fTOSSPercentage:=0;
END_IF

END_FUNCTION_BLOCK

// P_Machine
PROGRAM P_Machine
VAR_INPUT
	StationCount:				INT;
END_VAR
VAR
	_fbSystem:					FB_System;
	_iRunCount:					INT;
	_i:							INT;
END_VAR

IF _iRunCount<1 THEN
	_iRunCount:=_iRunCount+1;
	RETURN;
END_IF

_fbSystem(System:=G_stSystem,Error:=G_stError, Station:=ADR(G_arrStation) , StationCount:=StationCount );

P_Recipe();


FOR _i:=0 TO 20 BY 1 DO
	G_arrFbAxis[_i](Axis:=G_arrAxis[_i] , Data:=G_arrAxisData[_i] , Error:=G_stError , System:=G_stSystem );
END_FOR

FOR _i:=0 TO 50 BY 1 DO
	G_arrFbCylinder[_i](System:=G_stSystem , Cylinder:=G_arrCylinder[_i] , Data:=G_arrCylinderData[_i] , Error:=G_stError );
END_FOR

END_PROGRAM

// Axis/VISUs/CtrlAxis
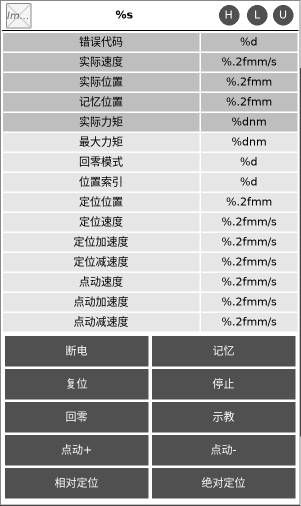
VISUALIZATION CtrlAxis  // 301x506
VAR_INPUT
	System:			REFERENCE TO ST_System;
	Axis:			REFERENCE TO ST_Axis;
	Data:			REFERENCE TO ST_AxisData;
END_VAR
    RoundedRectangle (0,391 300x115)
    RoundedRectangle (0,0 300x115)
    Rectangle (0,75 300x347)
    Rectangle (2,32 198x20), "错误代码", input disabled if: Axis.stLock.bShield
    Rectangle (200,32 98x20), "%d", text variable: Axis.stStatus.iErrorID, input disabled if: Axis.stLock.bShield
    Rectangle (2,52 198x20), "实际速度", input disabled if: Axis.stLock.bShield
    Rectangle (200,52 98x20), "%.2fmm/s", text variable: Axis.Axis_REF.NcToPlc.ActVelo, input disabled if: Axis.stLock.bShield
    Rectangle (2,72 198x20), "实际位置", input disabled if: Axis.stLock.bShield
    Rectangle (200,72 98x20), "%.2fmm", text variable: Axis.Axis_REF.NcToPlc.ActPos, input disabled if: Axis.stLock.bShield
    Rectangle (2,212 198x20), "定位速度", input disabled if: Axis.stLock.bShield
    Rectangle (200,212 98x20), "%.2fmm/s", text variable: Data.arrMoveVelocity[Axis.stControl.stMovePosition.iIndex], input disabled if: Axis.stLock.bShield
        OnMouseDown: write the text variable via VisuDialogs.Numpad
    Rectangle (2,232 198x20), "定位加速度", input disabled if: Axis.stLock.bShield
    Rectangle (2,172 198x20), "位置索引", input disabled if: Axis.stLock.bShield
    Rectangle (200,172 98x20), "%d", text variable: Axis.stControl.stMovePosition.iIndex, input disabled if: Axis.stLock.bShield
        OnMouseDown: write the text variable via VisuDialogs.Numpad, min 0, max 20
    Rectangle (200,232 98x20), "%.2fmm/s", text variable: Data.arrMoveAccelerated[Axis.stControl.stMovePosition.iIndex], input disabled if: Axis.stLock.bShield
        OnMouseDown: write the text variable via VisuDialogs.Numpad
    Rectangle (2,252 198x20), "定位减速度", input disabled if: Axis.stLock.bShield
    Rectangle (200,252 98x20), "%.2fmm/s", text variable: Data.arrMoveDeceleration[Axis.stControl.stMovePosition.iIndex], input disabled if: Axis.stLock.bShield
        OnMouseDown: write the text variable via VisuDialogs.Numpad
    Rectangle (2,272 198x20), "点动速度", input disabled if: Axis.stLock.bShield
    Rectangle (200,272 98x20), "%.2fmm/s", text variable: Data.fJogVelocity, input disabled if: Axis.stLock.bShield
        OnMouseDown: write the text variable via VisuDialogs.Numpad
    Rectangle (2,292 198x20), "点动加速度", input disabled if: Axis.stLock.bShield
    Rectangle (200,292 98x20), "%.2fmm/s", text variable: Data.fJogAccelerated, input disabled if: Axis.stLock.bShield
        OnMouseDown: write the text variable via VisuDialogs.Numpad
    Rectangle (2,312 198x20), "点动减速度", input disabled if: Axis.stLock.bShield
    Rectangle (200,312 98x20), "%.2fmm/s", text variable: Data.fJogDeceleration, input disabled if: Axis.stLock.bShield
        OnMouseDown: write the text variable via VisuDialogs.Numpad
    Rectangle (2,192 198x20), "定位位置", input disabled if: Axis.stLock.bShield
    Rectangle (200,192 98x20), "%.2fmm", text variable: Data.arrMovePosition[Axis.stControl.stMovePosition.iIndex], input disabled if: Axis.stLock.bShield
        OnMouseDown: write the text variable via VisuDialogs.Numpad
    Rectangle (2,92 198x20), "记忆位置", input disabled if: Axis.stLock.bShield
    Rectangle (200,92 98x20), "%.2fmm", text variable: Data.fMemoryPosition, input disabled if: Axis.stLock.bShield
    Rectangle (2,132 198x20), "最大力矩", input disabled if: Axis.stLock.bShield
    Rectangle (200,132 98x20), "%dnm", text variable: Data.stTorque.iSetTorque, input disabled if: Axis.stLock.bShield
        OnMouseDown: write the text variable via VisuDialogs.Numpad
    Rectangle (2,152 198x20), "回零模式", input disabled if: Axis.stLock.bShield
    RoundedRectangle (5,336 143x30), "断电", input disabled if: Axis.stLock.bShield
        toggle Axis.stControl.stClosePower.bManual
    RoundedRectangle (5,369 143x30), "复位", input disabled if: Axis.stLock.bShield
        tap Axis.stControl.stReset.bManual
    RoundedRectangle (152,369 143x30), "停止", input disabled if: Axis.stLock.bShield
        tap Axis.stControl.stStop.bManual
    RoundedRectangle (5,402 143x30), "回零", input disabled if: Axis.stLock.bShield
        tap Axis.stControl.stHome.bManual
    RoundedRectangle (152,402 143x30), "示教", input disabled if: Axis.stLock.bShield
        tap Axis.stControl.stTeach.bManual
    RoundedRectangle (5,435 143x30), "点动+", input disabled if: Axis.stLock.bShield
        tap Axis.stControl.stJog.stPositive.bManual
    RoundedRectangle (152,435 143x30), "点动-", input disabled if: Axis.stLock.bShield
        tap Axis.stControl.stJog.stNegative.bManual
    RoundedRectangle (5,468 143x30), "相对定位", input disabled if: Axis.stLock.bShield
        tap Axis.stControl.stMovePosition.stStartRel.bManual
    RoundedRectangle (152,468 143x30), "绝对定位", input disabled if: Axis.stLock.bShield
        tap Axis.stControl.stMovePosition.stStartAbs.bManual
    Line (2,30) (298,30)
    Rectangle (35,3 179x24), "%s", text variable: Axis.sName
    Ellipse (247,5 20x20), "L", colour toggle: Axis.stInput.bNegative
    Ellipse (273,5 20x20), "U", colour toggle: Axis.stInput.bPositive
    Line (300,68) (300,436)
    Line (0,60) (0,446)
    Image (6,3 25x25), image: ImagePool.axis
    Ellipse (219,5 20x20), "H", colour toggle: Axis.stStatus.bHomeDone
    Rectangle (200,152 98x20), "%d", text variable: Data.stMode.iHomeMode, input disabled if: Axis.stLock.bShield, text list: 'TextHomeMode', text index: Data.stMode.iHomeMode
        OnMouseDown: write the text variable via VisuDialogs.Numpad, min 0, max 9
    RoundedRectangle (152,336 143x30), "记忆", input disabled if: Axis.stLock.bShield OR Not Axis.stStatus.bMemoryPos
        tap Axis.stControl.stMoveMemory.bManual
    Rectangle (2,112 198x20), "实际力矩", input disabled if: Axis.stLock.bShield
    Rectangle (200,112 98x20), "%dnm", text variable: Data.stTorque.iGetTorque, input disabled if: Axis.stLock.bShield
END_VISUALIZATION

// Axis/VISUs/CtrlAxisGroup
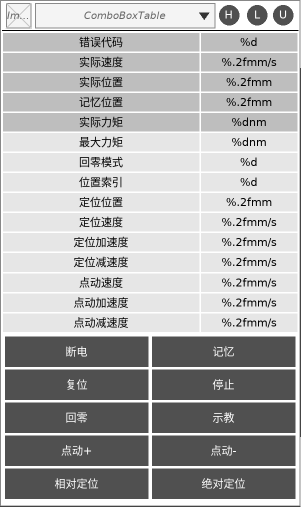
VISUALIZATION CtrlAxisGroup  // 301x507
VAR_INPUT
	System:						REFERENCE TO ST_System;
	Axis:						REFERENCE TO ARRAY[0..20] OF ST_Axis;
	Data:						REFERENCE TO ARRAY[0..20] OF ST_AxisData;
END_VAR
VAR
	_i:							INT;
END_VAR
    Frame (0,0 301x507)
        shows CtrlAxis(System := System, Axis := Axis[_i], Data := Data[_i])
    ComboBoxTable (35,3 180x25), variable: _i, data array: Axis
        p3854506369: Axis[INDEX].sName
        p1892666644: Axis[INDEX].stInput
        p338671338: Axis[INDEX].stLock
        p2170511999: Axis[INDEX].stStatus
        p3723444502: Axis[INDEX].stControl
        p1218418051: Axis[INDEX].Axis_REF
        p746581629: Axis[INDEX].arrInfo
END_VISUALIZATION

// Cylinder/VISUs/CtrlCylinder
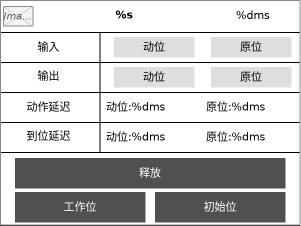
VISUALIZATION CtrlCylinder  // 301x226
VAR_INPUT
	System:							REFERENCE TO ST_System;
	Cylinder:						REFERENCE TO ST_Cylinder;
	CylinderData:					REFERENCE TO ST_CylinderData;
END_VAR
    RoundedRectangle (0,111 300x115)
    RoundedRectangle (0,0 300x115)
    Rectangle (0,34 300x115)
    Line (0,32) (300,32)
    Rectangle (35,3 179x24), "%s", text variable: Cylinder.arrInfo[System.stMode.eLanguage].sName, input disabled if: Cylinder.stLock.bShield
    Rectangle (218,3 70x25), "%dms", text variable: CylinderData.iAlarmTime, input disabled if: Cylinder.stLock.bShield
        OnMouseClick: write the text variable via VisuDialogs.Numpad
    Line (0,62) (300,62)
    Line (0,92) (300,92)
    Label (1,32 95x30), "输入"
    Label (1,61 95x30), "输出"
    Line (100,152) (100,32)
    RoundedRectangle (114,37 80x20), "动位", colour toggle: Cylinder.stInput.bWork, input disabled if: Cylinder.stLock.bShield
    RoundedRectangle (211,37 80x20), "原位", colour toggle: Cylinder.stInput.bHome, input disabled if: Cylinder.stLock.bShield
    RoundedRectangle (114,67 80x20), "动位", colour toggle: Cylinder.stOutput.bWork, input disabled if: Cylinder.stLock.bShield
    RoundedRectangle (211,67 80x20), "原位", colour toggle: Cylinder.stOutput.bHome, input disabled if: Cylinder.stLock.bShield
    RoundedRectangle (15,158 270x30), "释放", colour toggle: Cylinder.stLock.bOff OR Cylinder.stLock.bAll, input disabled if: Cylinder.stLock.bShield
        tap Cylinder.stControl.stOffRequest.bManual
    RoundedRectangle (15,192 130x30), "工作位", colour toggle: Cylinder.stLock.bWork OR Cylinder.stLock.bAll, input disabled if: Cylinder.stLock.bShield
        tap Cylinder.stControl.stWorkRequest.bManual
    RoundedRectangle (155,192 130x30), "初始位", colour toggle: Cylinder.stLock.bHome OR Cylinder.stLock.bAll, input disabled if: Cylinder.stLock.bShield
        tap Cylinder.stControl.stHomeRequest.bManual
    Line (300,154) (300,23)
    Line (0,152) (0,19)
    Image (3,6 30x20), image: ImagePool.Cylinder1
    Line (0,122) (300,122)
    Line (0,152) (300,152)
    Label (1,92 95x30), "动作延迟"
    Label (1,121 95x30), "到位延迟"
    RoundedRectangle (103,94 95x26), "动位:%dms", text variable: CylinderData.iWorkRequestTime, input disabled if: Cylinder.stLock.bShield
        OnMouseClick: write the text variable via Default
    RoundedRectangle (203,94 95x26), "原位:%dms", text variable: CylinderData.iHomeRequestTime, input disabled if: Cylinder.stLock.bShield
        OnMouseClick: write the text variable via Default
    RoundedRectangle (103,124 95x26), "动位:%dms", text variable: CylinderData.iWorkDone, input disabled if: Cylinder.stLock.bShield
        OnMouseClick: write the text variable via Default
    RoundedRectangle (203,124 95x26), "原位:%dms", text variable: CylinderData.iHomeDone, input disabled if: Cylinder.stLock.bShield
        OnMouseClick: write the text variable via Default
END_VISUALIZATION

// Cylinder/VISUs/CtrlCylinderGroup
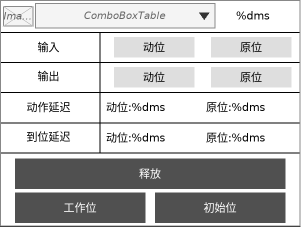
VISUALIZATION CtrlCylinderGroup  // 301x227
VAR_INPUT
	System:						REFERENCE TO ST_System;
	Cylinder:					REFERENCE TO ARRAY[0..50] OF ST_Cylinder;
	CylinderData:				REFERENCE TO ARRAY[0..50] OF ST_CylinderData;
END_VAR
VAR
	_i:							INT;
END_VAR
    Frame (0,0 301x227)
        shows CtrlCylinder(System := System, Cylinder := Cylinder[_i], CylinderData := CylinderData[_i])
    ComboBoxTable (35,3 180x25), variable: _i, data array: Cylinder
        p3854506369: Cylinder[INDEX].sName
        p1892666644: Cylinder[INDEX].stInput
        p338671338: Cylinder[INDEX].stOutput
        p2170511999: Cylinder[INDEX].stControl
        p3723444502: Cylinder[INDEX].stLock
        p1218418051: Cylinder[INDEX].stStatus
        p746581629: Cylinder[INDEX].arrInfo
END_VISUALIZATION

// Error/VISUs/CtrlError
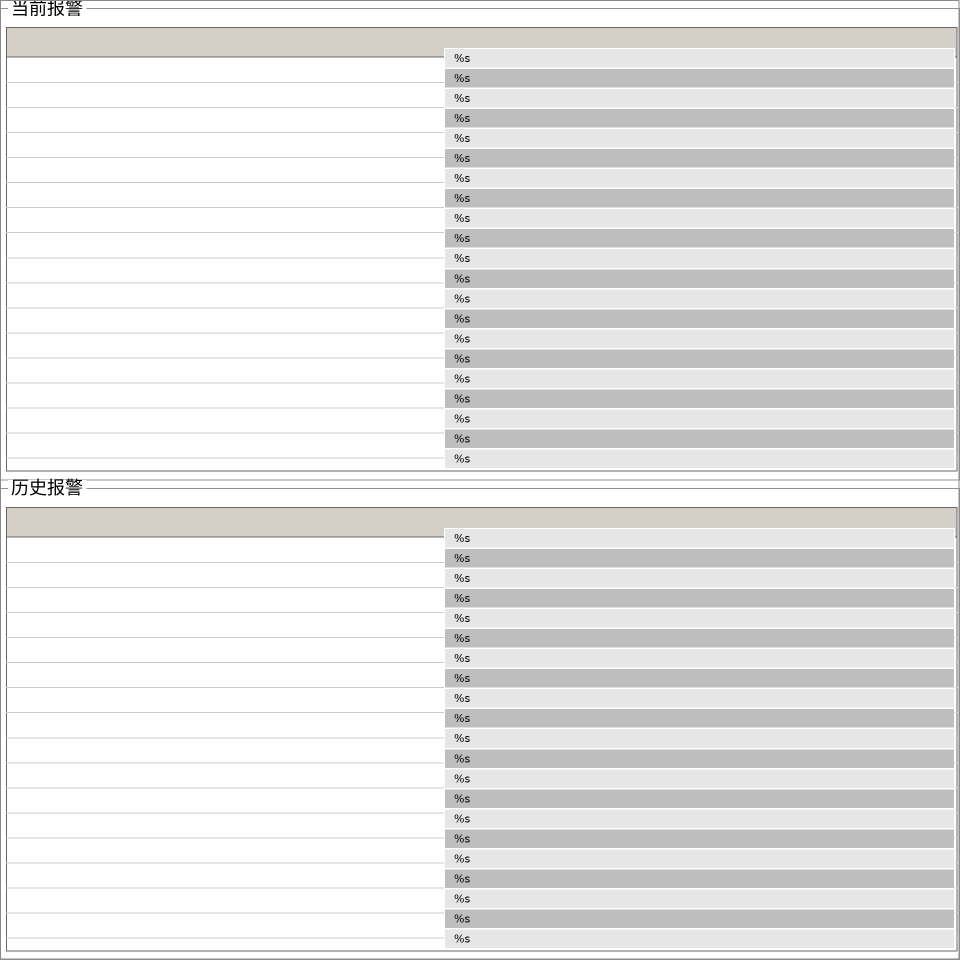
VISUALIZATION CtrlError  // 960x960
VAR_INPUT
	System:					REFERENCE TO ST_System;
	Error:					REFERENCE TO ST_Error;
END_VAR
    GroupBox (0,0 960x480), "当前报警"
        Frame (6,27 951x444)
            shows CtrlErrorGroup(System := System, Error := Error.stNow)
    GroupBox (0,480 960x480), "历史报警"
        Frame (6,27 951x444)
            shows CtrlErrorGroup(System := System, Error := Error.stHistory)
END_VISUALIZATION

// Error/VISUs/CtrlError1
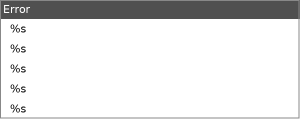
VISUALIZATION CtrlError1  // 300x119
VAR_INPUT
	System:					REFERENCE TO ST_System;
	Error:					REFERENCE TO ST_ErrorGroup;
END_VAR
    Rectangle (0,0 300x19), "Error"
    Rectangle (0,19 300x20), "%s", text variable: Error.arrInfo[0].arrMessage[System.stMode.eLanguage]
    Rectangle (0,39 300x20), "%s", text variable: Error.arrInfo[1].arrMessage[System.stMode.eLanguage]
    Rectangle (0,59 300x20), "%s", text variable: Error.arrInfo[2].arrMessage[System.stMode.eLanguage]
    Rectangle (0,79 300x20), "%s", text variable: Error.arrInfo[3].arrMessage[System.stMode.eLanguage]
    Rectangle (0,99 300x20), "%s", text variable: Error.arrInfo[4].arrMessage[System.stMode.eLanguage]
END_VISUALIZATION

